// TIA Portal V17 export
// export: Created 2023-02-13T11:16:18.7085922Z, ExportSetting WithDefaults, DisplayName Totally Integrated Automation Portal, DisplayVersion V17, DisplayName TIA Portal Openness, DisplayVersion V17, DisplayName TIA Portal Teamcenter Gateway, DisplayVersion V17, DisplayName TIA Portal Version Control Interface, DisplayVersion V17, DisplayName SINAMICS Startdrive Advanced, DisplayVersion V17, DisplayName SINAMICS Startdrive G130, G150, S120, S150, SINAMICS MV, S210, DisplayVersion V17, DisplayName SINAMICS Startdrive G110M, G120, G120C, G120D, G120P, G115D, DisplayVersion V17, DisplayName STEP 7 Professional, DisplayVersion V17, DisplayName STEP 7 Safety, DisplayVersion V17, DisplayName WinCC Professional, DisplayVersion V17
FUNCTION_BLOCK "IO_Valve_Blend30"   // FB26, LAD
{ S7_Optimized_Access := 'FALSE' }
VERSION : 0.1
// stored: AutoNumber true, IsIECCheckEnabled false, SetENOAutomatically false, UDAEnableTagReadback false
   VAR_INPUT
      "lock 1" : Bool;
      "lock 2" : Bool;
      "lock 3" : Bool;
      "lock 4" : Bool;
      init : Bool;
      reset : Bool;
      testing : Bool;
   END_VAR
   VAR
      "AV-30.01" : "Valve";
      "AV-30.02" : "Valve";
      "AV-30.03" : "Valve";
      "AV-30.04" : "Valve";
      "AV-30.05" : "Valve";
      "AV-30.06" : "Valve";
      "AV-30.07" : "Valve";
      "AV-30.08" : "Valve";
      "AV-30.09" : "Valve";
      "AV-30.10" : "Valve";
      "AV-30.11" : "Valve";
      "AV-30.12" : "Valve";
      "AV-30.13" : "Valve";
      "AV-30.14" : "Valve";
      "AV-30.15" : "Valve";
      "AV-30.16" : "Valve";
      "AV-30.17" : "Valve";
      "AV-30.18" : "Valve";
      "AV-30.19" : "Valve";
      "AV-30.20" : "Valve";
      "AV-30.21" : "Valve";
      "AV-30.22" : "Valve";
      "AV-30.23" : "Valve";
      "AV-30.24" : "Valve";
      "AV-30.25" : "Valve";
      "AV-30.26" : "Valve";
      "AV-30.27" : "Valve";
      "AV-30.28" : "Valve";
      "AV-30.29" : "Valve";
      "AV-30.30" : "Valve";
      "AV-30.31" : "Valve";
      "AV-30.32" : "Valve";
      "AV-30.33" : "Valve";
      "AV-30.34" : "Valve";
      "AV-30.35" : "Valve";
      "AV-30.36" : "Valve";
      "AV-30.41" : "Valve";
      "AV-30.42" : "Valve";
   END_VAR
BEGIN

REGION Network 2 (SCL): FB OPEN AND CLOSE VALVE T-30
   IF #testing THEN
       // Statement section IF
       #"AV-30.01".FB_OPEN := #"AV-30.01".QCMD_OP;
       #"AV-30.01".FB_CLOSE := NOT #"AV-30.01".QCMD_OP;
       #"AV-30.02".FB_OPEN := #"AV-30.02".QCMD_OP;
       #"AV-30.02".FB_CLOSE := NOT #"AV-30.02".QCMD_OP;
       #"AV-30.03".FB_OPEN := #"AV-30.03".QCMD_OP;
       #"AV-30.03".FB_CLOSE := NOT #"AV-30.03".QCMD_OP;
       #"AV-30.04".FB_OPEN := #"AV-30.04".QCMD_OP;
       #"AV-30.04".FB_CLOSE := NOT #"AV-30.04".QCMD_OP;
       #"AV-30.05".FB_OPEN := #"AV-30.05".QCMD_OP;
       #"AV-30.05".FB_CLOSE := NOT #"AV-30.05".QCMD_OP;
       #"AV-30.06".FB_OPEN := #"AV-30.06".QCMD_OP;
       #"AV-30.06".FB_CLOSE := NOT #"AV-30.06".QCMD_OP;
       #"AV-30.07".FB_OPEN := #"AV-30.07".QCMD_OP;
       #"AV-30.07".FB_CLOSE := NOT #"AV-30.07".QCMD_OP;
       #"AV-30.08".FB_OPEN := #"AV-30.08".QCMD_OP;
       #"AV-30.08".FB_CLOSE := NOT #"AV-30.08".QCMD_OP;
       #"AV-30.09".FB_OPEN := #"AV-30.09".QCMD_OP;
       #"AV-30.09".FB_CLOSE := NOT #"AV-30.09".QCMD_OP;
       #"AV-30.10".FB_OPEN := #"AV-30.10".QCMD_OP;
       #"AV-30.10".FB_CLOSE := NOT #"AV-30.10".QCMD_OP;
       #"AV-30.11".FB_OPEN := #"AV-30.11".QCMD_OP;
       #"AV-30.11".FB_CLOSE := NOT #"AV-30.11".QCMD_OP;
       #"AV-30.12".FB_OPEN := #"AV-30.12".QCMD_OP;
       #"AV-30.12".FB_CLOSE := NOT #"AV-30.12".QCMD_OP;
       #"AV-30.13".FB_OPEN := #"AV-30.13".QCMD_OP;
       #"AV-30.13".FB_CLOSE := NOT #"AV-30.13".QCMD_OP;
       #"AV-30.14".FB_OPEN := #"AV-30.14".QCMD_OP;
       #"AV-30.14".FB_CLOSE := NOT #"AV-30.14".QCMD_OP;
       #"AV-30.15".FB_OPEN := #"AV-30.15".QCMD_OP;
       #"AV-30.15".FB_CLOSE := NOT #"AV-30.15".QCMD_OP;
       #"AV-30.16".FB_OPEN := #"AV-30.16".QCMD_OP;
       #"AV-30.16".FB_CLOSE := NOT #"AV-30.16".QCMD_OP;
       #"AV-30.17".FB_OPEN := #"AV-30.17".QCMD_OP;
       #"AV-30.17".FB_CLOSE := NOT #"AV-30.17".QCMD_OP;
       #"AV-30.18".FB_OPEN := #"AV-30.18".QCMD_OP;
       #"AV-30.18".FB_CLOSE := NOT #"AV-30.18".QCMD_OP;
       #"AV-30.19".FB_OPEN := #"AV-30.19".QCMD_OP;
       #"AV-30.19".FB_CLOSE := NOT #"AV-30.19".QCMD_OP;
       #"AV-30.20".FB_OPEN := #"AV-30.20".QCMD_OP;
       #"AV-30.20".FB_CLOSE := NOT #"AV-30.20".QCMD_OP;
       #"AV-30.21".FB_OPEN := #"AV-30.21".QCMD_OP;
       #"AV-30.21".FB_CLOSE := NOT #"AV-30.21".QCMD_OP;
       #"AV-30.22".FB_OPEN := #"AV-30.22".QCMD_OP;
       #"AV-30.22".FB_CLOSE := NOT #"AV-30.22".QCMD_OP;
       #"AV-30.23".FB_OPEN := #"AV-30.23".QCMD_OP;
       #"AV-30.23".FB_CLOSE := NOT #"AV-30.23".QCMD_OP;
       #"AV-30.24".FB_OPEN := #"AV-30.24".QCMD_OP;
       #"AV-30.24".FB_CLOSE := NOT #"AV-30.24".QCMD_OP;
       #"AV-30.25".FB_OPEN := #"AV-30.25".QCMD_OP;
       #"AV-30.25".FB_CLOSE := NOT #"AV-30.25".QCMD_OP;
       #"AV-30.26".FB_OPEN := #"AV-30.26".QCMD_OP;
       #"AV-30.26".FB_CLOSE := NOT #"AV-30.26".QCMD_OP;
       #"AV-30.27".FB_OPEN := #"AV-30.27".QCMD_OP;
       #"AV-30.27".FB_CLOSE := NOT #"AV-30.27".QCMD_OP;
       #"AV-30.28".FB_OPEN := #"AV-30.28".QCMD_OP;
       #"AV-30.28".FB_CLOSE := NOT #"AV-30.28".QCMD_OP;
       #"AV-30.29".FB_OPEN := #"AV-30.29".QCMD_OP;
       #"AV-30.29".FB_CLOSE := NOT #"AV-30.29".QCMD_OP;
       #"AV-30.30".FB_OPEN := #"AV-30.30".QCMD_OP;
       #"AV-30.30".FB_CLOSE := NOT #"AV-30.30".QCMD_OP;
       #"AV-30.31".FB_OPEN := #"AV-30.31".QCMD_OP;
       #"AV-30.31".FB_CLOSE := NOT #"AV-30.31".QCMD_OP;
       #"AV-30.32".FB_OPEN := #"AV-30.32".QCMD_OP;
       #"AV-30.32".FB_CLOSE := NOT #"AV-30.32".QCMD_OP;
       #"AV-30.33".FB_OPEN := #"AV-30.33".QCMD_OP;
       #"AV-30.33".FB_CLOSE := NOT #"AV-30.33".QCMD_OP;
       #"AV-30.34".FB_OPEN := #"AV-30.34".QCMD_OP;
       #"AV-30.34".FB_CLOSE := NOT #"AV-30.34".QCMD_OP;
       #"AV-30.35".FB_OPEN := #"AV-30.35".QCMD_OP;
       #"AV-30.35".FB_CLOSE := NOT #"AV-30.35".QCMD_OP;
       #"AV-30.36".FB_OPEN := #"AV-30.36".QCMD_OP;
       #"AV-30.36".FB_CLOSE := NOT #"AV-30.36".QCMD_OP;
       #"AV-30.41".FB_OPEN := #"AV-30.41".QCMD_OP;
       #"AV-30.41".FB_CLOSE := NOT #"AV-30.41".QCMD_OP;
       #"AV-30.42".FB_OPEN := #"AV-30.42".QCMD_OP;
       #"AV-30.42".FB_CLOSE := NOT #"AV-30.42".QCMD_OP;
   ELSE
       // Statement section ELSE
       #"AV-30.01".FB_OPEN := #"AV-30.01".QCMD_OP;
       #"AV-30.01".FB_CLOSE := NOT #"AV-30.01".QCMD_OP;
       #"AV-30.02".FB_OPEN := NOT "ZSC-30.02";
       #"AV-30.02".FB_CLOSE := "ZSC-30.02";
       #"AV-30.03".FB_OPEN := NOT "ZSC-30.03";
       #"AV-30.03".FB_CLOSE := "ZSC-30.03";
       #"AV-30.04".FB_OPEN := #"AV-30.04".QCMD_OP;
       #"AV-30.04".FB_CLOSE := NOT #"AV-30.04".QCMD_OP;
       #"AV-30.05".FB_OPEN := NOT "ZSC-30.05";
       #"AV-30.05".FB_CLOSE := "ZSC-30.05";
       #"AV-30.06".FB_OPEN := NOT "ZSC-30.06";
       #"AV-30.06".FB_CLOSE := "ZSC-30.06";
       #"AV-30.07".FB_OPEN := #"AV-30.07".QCMD_OP;
       #"AV-30.07".FB_CLOSE := NOT #"AV-30.07".QCMD_OP;
       #"AV-30.08".FB_OPEN := NOT "ZSC-30.08";
       #"AV-30.08".FB_CLOSE := "ZSC-30.08";
       #"AV-30.09".FB_OPEN := NOT "ZSC-30.09";
       #"AV-30.09".FB_CLOSE := "ZSC-30.09";
       #"AV-30.10".FB_OPEN := #"AV-30.10".QCMD_OP;
       #"AV-30.10".FB_CLOSE := NOT #"AV-30.10".QCMD_OP;
       #"AV-30.11".FB_OPEN := NOT "ZSC-30.11";
       #"AV-30.11".FB_CLOSE := "ZSC-30.11";
       #"AV-30.12".FB_OPEN := #"AV-30.12".QCMD_OP;
       #"AV-30.12".FB_CLOSE := NOT #"AV-30.12".QCMD_OP;
       #"AV-30.13".FB_OPEN := #"AV-30.13".QCMD_OP;
       #"AV-30.13".FB_CLOSE := NOT #"AV-30.13".QCMD_OP;
       #"AV-30.14".FB_OPEN := NOT "ZSC-30.14";
       #"AV-30.14".FB_CLOSE := "ZSC-30.14";
       #"AV-30.15".FB_OPEN := #"AV-30.15".QCMD_OP;
       #"AV-30.15".FB_CLOSE := NOT #"AV-30.15".QCMD_OP;
       #"AV-30.16".FB_OPEN := #"AV-30.16".QCMD_OP;
       #"AV-30.16".FB_CLOSE := NOT #"AV-30.16".QCMD_OP;
       #"AV-30.17".FB_OPEN := NOT "ZSC-30.17";
       #"AV-30.17".FB_CLOSE := "ZSC-30.17";
       #"AV-30.18".FB_OPEN := #"AV-30.18".QCMD_OP;
       #"AV-30.18".FB_CLOSE := NOT #"AV-30.18".QCMD_OP;
       #"AV-30.19".FB_OPEN := #"AV-30.19".QCMD_OP;
       #"AV-30.19".FB_CLOSE := NOT #"AV-30.19".QCMD_OP;
       #"AV-30.20".FB_OPEN := NOT "ZSC-30.20";
       #"AV-30.20".FB_CLOSE := "ZSC-30.20";
       #"AV-30.21".FB_OPEN := NOT "ZSC-30.21";
       #"AV-30.21".FB_CLOSE := "ZSC-30.21";
       #"AV-30.22".FB_OPEN := #"AV-30.22".QCMD_OP;
       #"AV-30.22".FB_CLOSE := NOT #"AV-30.22".QCMD_OP;
       #"AV-30.23".FB_OPEN := NOT "ZSC-30.23";
       #"AV-30.23".FB_CLOSE := "ZSC-30.23";
       #"AV-30.24".FB_OPEN := NOT "ZSC-30.24";
       #"AV-30.24".FB_CLOSE := "ZSC-30.24";
       #"AV-30.25".FB_OPEN := NOT "ZSC-30.25";
       #"AV-30.25".FB_CLOSE := "ZSC-30.25";
       #"AV-30.26".FB_OPEN := #"AV-30.26".QCMD_OP;
       #"AV-30.26".FB_CLOSE := NOT #"AV-30.26".QCMD_OP;
       #"AV-30.27".FB_OPEN := NOT "ZSC-30.27";
       #"AV-30.27".FB_CLOSE := "ZSC-30.27";
       #"AV-30.28".FB_OPEN := NOT "ZSC-30.28";
       #"AV-30.28".FB_CLOSE := "ZSC-30.28";
       #"AV-30.29".FB_OPEN := #"AV-30.29".QCMD_OP;
       #"AV-30.29".FB_CLOSE := NOT #"AV-30.29".QCMD_OP;
       #"AV-30.30".FB_OPEN := #"AV-30.30".QCMD_OP;
       #"AV-30.30".FB_CLOSE := NOT #"AV-30.30".QCMD_OP;
       #"AV-30.31".FB_OPEN := NOT "ZSC-30.31";
       #"AV-30.31".FB_CLOSE := "ZSC-30.31";
       #"AV-30.32".FB_OPEN := NOT "ZSC-30.32";
       #"AV-30.32".FB_CLOSE := "ZSC-30.32";
       #"AV-30.33".FB_OPEN := NOT "ZSC-30.33";
       #"AV-30.33".FB_CLOSE := "ZSC-30.33";
       #"AV-30.34".FB_OPEN := NOT "ZSC-30.34";
       #"AV-30.34".FB_CLOSE := "ZSC-30.34";
       #"AV-30.35".FB_OPEN := NOT "ZSC-30.35";
       #"AV-30.35".FB_CLOSE := "ZSC-30.35";
       #"AV-30.36".FB_OPEN := NOT "ZSC-30.36";
       #"AV-30.36".FB_CLOSE := "ZSC-30.36";
       #"AV-30.41".FB_OPEN := #"AV-30.41".QCMD_OP;
       #"AV-30.41".FB_CLOSE := NOT #"AV-30.41".QCMD_OP;
       #"AV-30.42".FB_OPEN := #"AV-30.42".QCMD_OP;
       #"AV-30.42".FB_CLOSE := NOT #"AV-30.42".QCMD_OP;
   END_IF;
END_REGION

NETWORK
TITLE = FB MONITORING TIME VALVE T-30
// FB OPEN TIME
      L     T#20s;
      T     #"AV-30.01".MON_T;
      T     #"AV-30.02".MON_T;
      T     #"AV-30.03".MON_T;
      T     #"AV-30.04".MON_T;
      T     #"AV-30.05".MON_T;
      T     #"AV-30.06".MON_T;
      T     #"AV-30.07".MON_T;
      T     #"AV-30.08".MON_T;
      T     #"AV-30.09".MON_T;
      T     #"AV-30.10".MON_T;
      T     #"AV-30.11".MON_T;
      T     #"AV-30.12".MON_T;
      T     #"AV-30.13".MON_T;
      T     #"AV-30.14".MON_T;
      T     #"AV-30.15".MON_T;
      T     #"AV-30.16".MON_T;
      T     #"AV-30.17".MON_T;
      T     #"AV-30.18".MON_T;
      T     #"AV-30.19".MON_T;
      T     #"AV-30.20".MON_T;
      T     #"AV-30.21".MON_T;
      T     #"AV-30.22".MON_T;
      T     #"AV-30.23".MON_T;
      T     #"AV-30.24".MON_T;
      T     #"AV-30.25".MON_T;
      T     #"AV-30.26".MON_T;
      T     #"AV-30.27".MON_T;
      T     #"AV-30.28".MON_T;
      T     #"AV-30.29".MON_T;
      T     #"AV-30.30".MON_T;
      T     #"AV-30.31".MON_T;
      T     #"AV-30.32".MON_T;
      T     #"AV-30.33".MON_T;
      T     #"AV-30.34".MON_T;
      T     #"AV-30.35".MON_T;
      T     #"AV-30.36".MON_T;
      T     #"AV-30.41".MON_T;
      T     #"AV-30.42".MON_T;
// FB CLOSE TIME
      L     T#20s;
      T     #"AV-30.01".MON_T_CLOSE;
      T     #"AV-30.02".MON_T_CLOSE;
      T     #"AV-30.03".MON_T_CLOSE;
      T     #"AV-30.04".MON_T_CLOSE;
      T     #"AV-30.05".MON_T_CLOSE;
      T     #"AV-30.06".MON_T_CLOSE;
      T     #"AV-30.07".MON_T_CLOSE;
      T     #"AV-30.08".MON_T_CLOSE;
      T     #"AV-30.09".MON_T_CLOSE;
      T     #"AV-30.10".MON_T_CLOSE;
      T     #"AV-30.11".MON_T_CLOSE;
      T     #"AV-30.12".MON_T_CLOSE;
      T     #"AV-30.13".MON_T_CLOSE;
      T     #"AV-30.14".MON_T_CLOSE;
      T     #"AV-30.15".MON_T_CLOSE;
      T     #"AV-30.16".MON_T_CLOSE;
      T     #"AV-30.17".MON_T_CLOSE;
      T     #"AV-30.18".MON_T_CLOSE;
      T     #"AV-30.19".MON_T_CLOSE;
      T     #"AV-30.20".MON_T_CLOSE;
      T     #"AV-30.21".MON_T_CLOSE;
      T     #"AV-30.22".MON_T_CLOSE;
      T     #"AV-30.23".MON_T_CLOSE;
      T     #"AV-30.24".MON_T_CLOSE;
      T     #"AV-30.25".MON_T_CLOSE;
      T     #"AV-30.26".MON_T_CLOSE;
      T     #"AV-30.27".MON_T_CLOSE;
      T     #"AV-30.28".MON_T_CLOSE;
      T     #"AV-30.29".MON_T_CLOSE;
      T     #"AV-30.30".MON_T_CLOSE;
      T     #"AV-30.31".MON_T_CLOSE;
      T     #"AV-30.32".MON_T_CLOSE;
      T     #"AV-30.33".MON_T_CLOSE;
      T     #"AV-30.34".MON_T_CLOSE;
      T     #"AV-30.35".MON_T_CLOSE;
      T     #"AV-30.36".MON_T_CLOSE;
      T     #"AV-30.41".MON_T_CLOSE;
      T     #"AV-30.42".MON_T_CLOSE;

REGION Network 4: AV-30.01
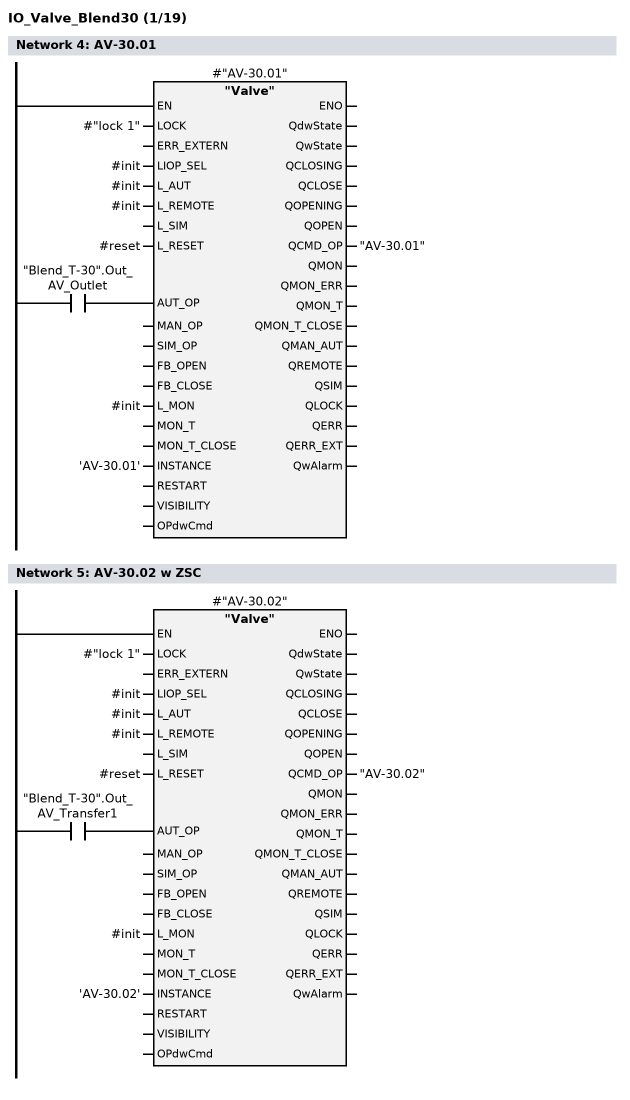
   RUNG wire#powerrail
      #"AV-30.01"(AUT_OP := wire#w1, LOCK := #"lock 1", ERR_EXTERN :=, LIOP_SEL := #init, L_AUT := #init, L_REMOTE := #init, L_SIM :=, L_RESET := #reset, MAN_OP :=, SIM_OP :=, FB_OPEN :=, FB_CLOSE :=, L_MON := #init, MON_T :=, MON_T_CLOSE :=, INSTANCE := 'AV-30.01', RESTART :=, VISIBILITY :=, OPdwCmd :=, QdwState =>, QwState =>, QCLOSING =>, QCLOSE =>, QOPENING =>, QOPEN =>, QCMD_OP => "AV-30.01", QMON =>, QMON_ERR =>, QMON_T =>, QMON_T_CLOSE =>, QMAN_AUT =>, QREMOTE =>, QSIM =>, QLOCK =>, QERR =>, QERR_EXT =>, QwAlarm =>)
   END_RUNG
   RUNG wire#powerrail
      Contact( "Blend_T-30".Out_AV_Outlet )
   END_RUNG wire#w1
   // the same network as SCL:
   #"AV-30.01"(LOCK := #"lock 1",   // "Valve"
               LIOP_SEL := #init,
               L_AUT := #init,
               L_REMOTE := #init,
               L_RESET := #reset,
               AUT_OP := "Blend_T-30".Out_AV_Outlet,
               L_MON := #init,
               INSTANCE := 'AV-30.01',
               QCMD_OP => "AV-30.01");
END_REGION

REGION Network 5: AV-30.02 w ZSC
   RUNG wire#powerrail
      #"AV-30.02"(AUT_OP := wire#w1, LOCK := #"lock 1", ERR_EXTERN :=, LIOP_SEL := #init, L_AUT := #init, L_REMOTE := #init, L_SIM :=, L_RESET := #reset, MAN_OP :=, SIM_OP :=, FB_OPEN :=, FB_CLOSE :=, L_MON := #init, MON_T :=, MON_T_CLOSE :=, INSTANCE := 'AV-30.02', RESTART :=, VISIBILITY :=, OPdwCmd :=, QdwState =>, QwState =>, QCLOSING =>, QCLOSE =>, QOPENING =>, QOPEN =>, QCMD_OP => "AV-30.02", QMON =>, QMON_ERR =>, QMON_T =>, QMON_T_CLOSE =>, QMAN_AUT =>, QREMOTE =>, QSIM =>, QLOCK =>, QERR =>, QERR_EXT =>, QwAlarm =>)
   END_RUNG
   RUNG wire#powerrail
      Contact( "Blend_T-30".Out_AV_Transfer1 )
   END_RUNG wire#w1
   // the same network as SCL:
   #"AV-30.02"(LOCK := #"lock 1",   // "Valve"
               LIOP_SEL := #init,
               L_AUT := #init,
               L_REMOTE := #init,
               L_RESET := #reset,
               AUT_OP := "Blend_T-30".Out_AV_Transfer1,
               L_MON := #init,
               INSTANCE := 'AV-30.02',
               QCMD_OP => "AV-30.02");
END_REGION

REGION Network 6: AV-30.03 w ZSC
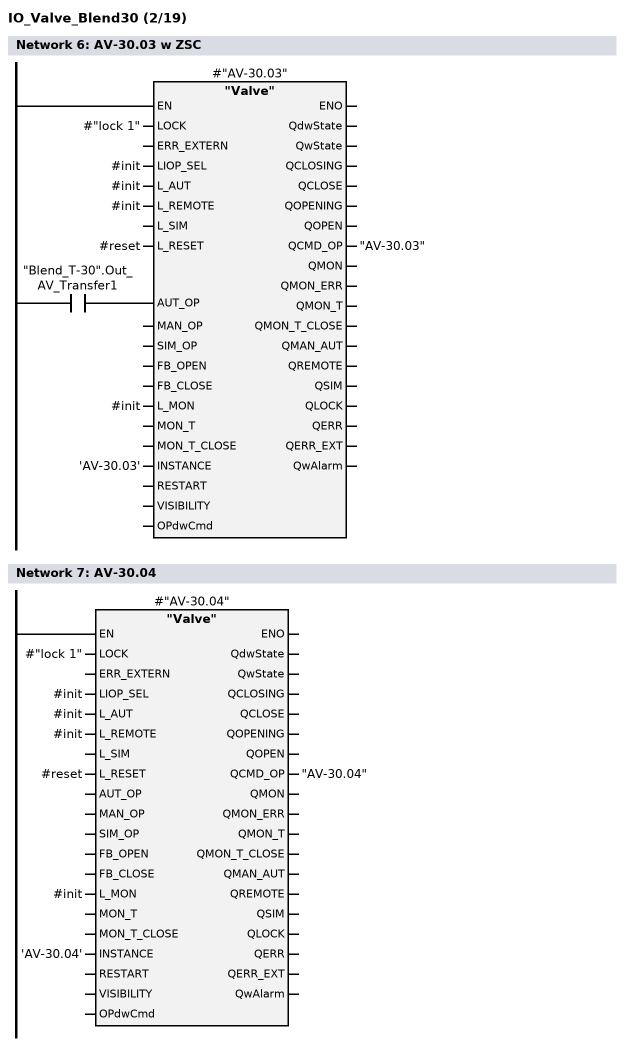
   RUNG wire#powerrail
      #"AV-30.03"(AUT_OP := wire#w1, LOCK := #"lock 1", ERR_EXTERN :=, LIOP_SEL := #init, L_AUT := #init, L_REMOTE := #init, L_SIM :=, L_RESET := #reset, MAN_OP :=, SIM_OP :=, FB_OPEN :=, FB_CLOSE :=, L_MON := #init, MON_T :=, MON_T_CLOSE :=, INSTANCE := 'AV-30.03', RESTART :=, VISIBILITY :=, OPdwCmd :=, QdwState =>, QwState =>, QCLOSING =>, QCLOSE =>, QOPENING =>, QOPEN =>, QCMD_OP => "AV-30.03", QMON =>, QMON_ERR =>, QMON_T =>, QMON_T_CLOSE =>, QMAN_AUT =>, QREMOTE =>, QSIM =>, QLOCK =>, QERR =>, QERR_EXT =>, QwAlarm =>)
   END_RUNG
   RUNG wire#powerrail
      Contact( "Blend_T-30".Out_AV_Transfer1 )
   END_RUNG wire#w1
   // the same network as SCL:
   #"AV-30.03"(LOCK := #"lock 1",   // "Valve"
               LIOP_SEL := #init,
               L_AUT := #init,
               L_REMOTE := #init,
               L_RESET := #reset,
               AUT_OP := "Blend_T-30".Out_AV_Transfer1,
               L_MON := #init,
               INSTANCE := 'AV-30.03',
               QCMD_OP => "AV-30.03");
END_REGION

REGION Network 7: AV-30.04
   RUNG wire#powerrail
      #"AV-30.04"(LOCK := #"lock 1", ERR_EXTERN :=, LIOP_SEL := #init, L_AUT := #init, L_REMOTE := #init, L_SIM :=, L_RESET := #reset, AUT_OP :=, MAN_OP :=, SIM_OP :=, FB_OPEN :=, FB_CLOSE :=, L_MON := #init, MON_T :=, MON_T_CLOSE :=, INSTANCE := 'AV-30.04', RESTART :=, VISIBILITY :=, OPdwCmd :=, QdwState =>, QwState =>, QCLOSING =>, QCLOSE =>, QOPENING =>, QOPEN =>, QCMD_OP => "AV-30.04", QMON =>, QMON_ERR =>, QMON_T =>, QMON_T_CLOSE =>, QMAN_AUT =>, QREMOTE =>, QSIM =>, QLOCK =>, QERR =>, QERR_EXT =>, QwAlarm =>)
   END_RUNG
   // the same network as SCL:
   #"AV-30.04"(LOCK := #"lock 1",   // "Valve"
               LIOP_SEL := #init,
               L_AUT := #init,
               L_REMOTE := #init,
               L_RESET := #reset,
               L_MON := #init,
               INSTANCE := 'AV-30.04',
               QCMD_OP => "AV-30.04");
END_REGION

REGION Network 8: AV-30.05 w ZSC
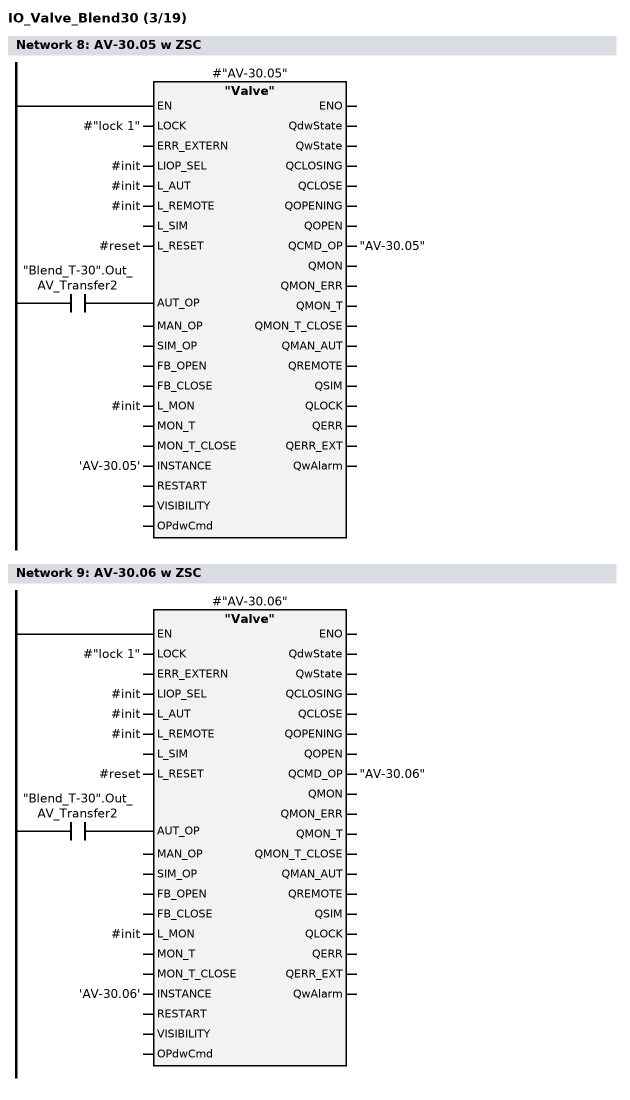
   RUNG wire#powerrail
      #"AV-30.05"(AUT_OP := wire#w1, LOCK := #"lock 1", ERR_EXTERN :=, LIOP_SEL := #init, L_AUT := #init, L_REMOTE := #init, L_SIM :=, L_RESET := #reset, MAN_OP :=, SIM_OP :=, FB_OPEN :=, FB_CLOSE :=, L_MON := #init, MON_T :=, MON_T_CLOSE :=, INSTANCE := 'AV-30.05', RESTART :=, VISIBILITY :=, OPdwCmd :=, QdwState =>, QwState =>, QCLOSING =>, QCLOSE =>, QOPENING =>, QOPEN =>, QCMD_OP => "AV-30.05", QMON =>, QMON_ERR =>, QMON_T =>, QMON_T_CLOSE =>, QMAN_AUT =>, QREMOTE =>, QSIM =>, QLOCK =>, QERR =>, QERR_EXT =>, QwAlarm =>)
   END_RUNG
   RUNG wire#powerrail
      Contact( "Blend_T-30".Out_AV_Transfer2 )
   END_RUNG wire#w1
   // the same network as SCL:
   #"AV-30.05"(LOCK := #"lock 1",   // "Valve"
               LIOP_SEL := #init,
               L_AUT := #init,
               L_REMOTE := #init,
               L_RESET := #reset,
               AUT_OP := "Blend_T-30".Out_AV_Transfer2,
               L_MON := #init,
               INSTANCE := 'AV-30.05',
               QCMD_OP => "AV-30.05");
END_REGION

REGION Network 9: AV-30.06 w ZSC
   RUNG wire#powerrail
      #"AV-30.06"(AUT_OP := wire#w1, LOCK := #"lock 1", ERR_EXTERN :=, LIOP_SEL := #init, L_AUT := #init, L_REMOTE := #init, L_SIM :=, L_RESET := #reset, MAN_OP :=, SIM_OP :=, FB_OPEN :=, FB_CLOSE :=, L_MON := #init, MON_T :=, MON_T_CLOSE :=, INSTANCE := 'AV-30.06', RESTART :=, VISIBILITY :=, OPdwCmd :=, QdwState =>, QwState =>, QCLOSING =>, QCLOSE =>, QOPENING =>, QOPEN =>, QCMD_OP => "AV-30.06", QMON =>, QMON_ERR =>, QMON_T =>, QMON_T_CLOSE =>, QMAN_AUT =>, QREMOTE =>, QSIM =>, QLOCK =>, QERR =>, QERR_EXT =>, QwAlarm =>)
   END_RUNG
   RUNG wire#powerrail
      Contact( "Blend_T-30".Out_AV_Transfer2 )
   END_RUNG wire#w1
   // the same network as SCL:
   #"AV-30.06"(LOCK := #"lock 1",   // "Valve"
               LIOP_SEL := #init,
               L_AUT := #init,
               L_REMOTE := #init,
               L_RESET := #reset,
               AUT_OP := "Blend_T-30".Out_AV_Transfer2,
               L_MON := #init,
               INSTANCE := 'AV-30.06',
               QCMD_OP => "AV-30.06");
END_REGION

REGION Network 10: AV-30.07
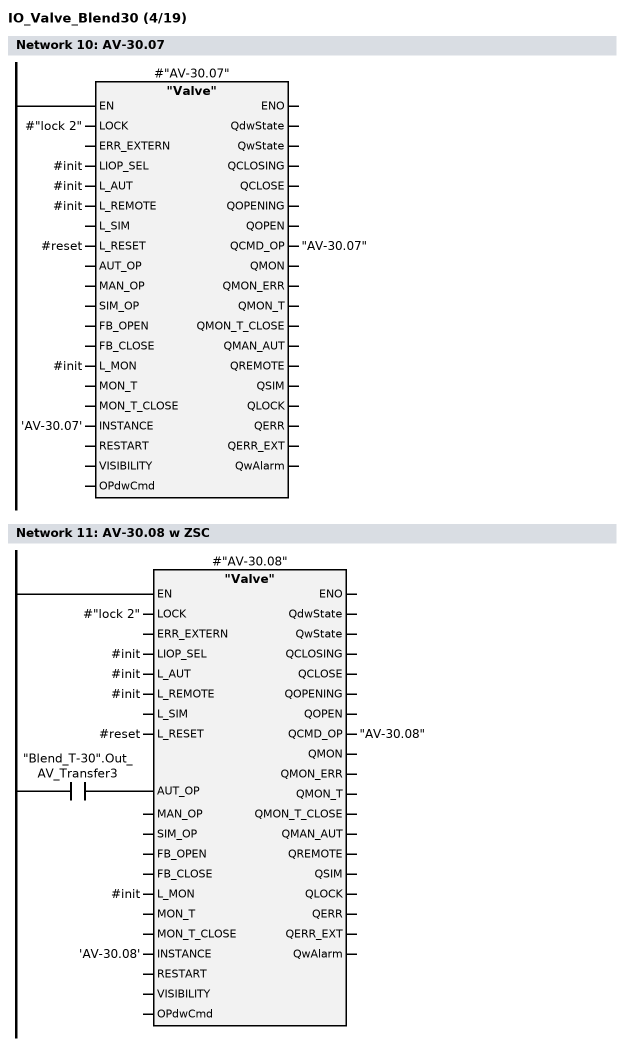
   RUNG wire#powerrail
      #"AV-30.07"(LOCK := #"lock 2", ERR_EXTERN :=, LIOP_SEL := #init, L_AUT := #init, L_REMOTE := #init, L_SIM :=, L_RESET := #reset, AUT_OP :=, MAN_OP :=, SIM_OP :=, FB_OPEN :=, FB_CLOSE :=, L_MON := #init, MON_T :=, MON_T_CLOSE :=, INSTANCE := 'AV-30.07', RESTART :=, VISIBILITY :=, OPdwCmd :=, QdwState =>, QwState =>, QCLOSING =>, QCLOSE =>, QOPENING =>, QOPEN =>, QCMD_OP => "AV-30.07", QMON =>, QMON_ERR =>, QMON_T =>, QMON_T_CLOSE =>, QMAN_AUT =>, QREMOTE =>, QSIM =>, QLOCK =>, QERR =>, QERR_EXT =>, QwAlarm =>)
   END_RUNG
   // the same network as SCL:
   #"AV-30.07"(LOCK := #"lock 2",   // "Valve"
               LIOP_SEL := #init,
               L_AUT := #init,
               L_REMOTE := #init,
               L_RESET := #reset,
               L_MON := #init,
               INSTANCE := 'AV-30.07',
               QCMD_OP => "AV-30.07");
END_REGION

REGION Network 11: AV-30.08 w ZSC
   RUNG wire#powerrail
      #"AV-30.08"(AUT_OP := wire#w1, LOCK := #"lock 2", ERR_EXTERN :=, LIOP_SEL := #init, L_AUT := #init, L_REMOTE := #init, L_SIM :=, L_RESET := #reset, MAN_OP :=, SIM_OP :=, FB_OPEN :=, FB_CLOSE :=, L_MON := #init, MON_T :=, MON_T_CLOSE :=, INSTANCE := 'AV-30.08', RESTART :=, VISIBILITY :=, OPdwCmd :=, QdwState =>, QwState =>, QCLOSING =>, QCLOSE =>, QOPENING =>, QOPEN =>, QCMD_OP => "AV-30.08", QMON =>, QMON_ERR =>, QMON_T =>, QMON_T_CLOSE =>, QMAN_AUT =>, QREMOTE =>, QSIM =>, QLOCK =>, QERR =>, QERR_EXT =>, QwAlarm =>)
   END_RUNG
   RUNG wire#powerrail
      Contact( "Blend_T-30".Out_AV_Transfer3 )
   END_RUNG wire#w1
   // the same network as SCL:
   #"AV-30.08"(LOCK := #"lock 2",   // "Valve"
               LIOP_SEL := #init,
               L_AUT := #init,
               L_REMOTE := #init,
               L_RESET := #reset,
               AUT_OP := "Blend_T-30".Out_AV_Transfer3,
               L_MON := #init,
               INSTANCE := 'AV-30.08',
               QCMD_OP => "AV-30.08");
END_REGION

REGION Network 12: AV-30.09 w ZSC
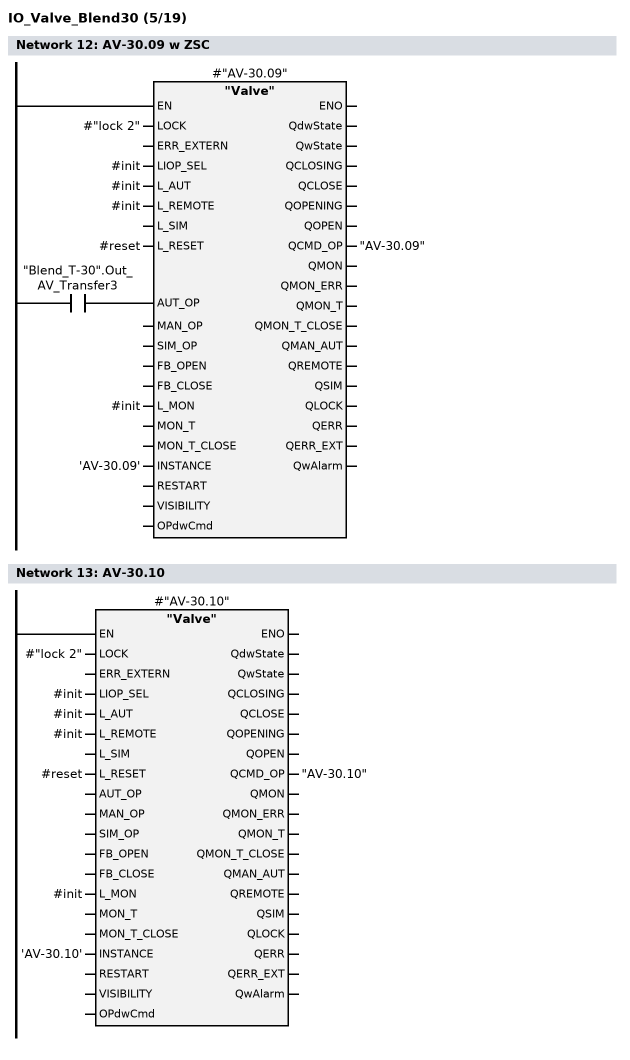
   RUNG wire#powerrail
      #"AV-30.09"(AUT_OP := wire#w1, LOCK := #"lock 2", ERR_EXTERN :=, LIOP_SEL := #init, L_AUT := #init, L_REMOTE := #init, L_SIM :=, L_RESET := #reset, MAN_OP :=, SIM_OP :=, FB_OPEN :=, FB_CLOSE :=, L_MON := #init, MON_T :=, MON_T_CLOSE :=, INSTANCE := 'AV-30.09', RESTART :=, VISIBILITY :=, OPdwCmd :=, QdwState =>, QwState =>, QCLOSING =>, QCLOSE =>, QOPENING =>, QOPEN =>, QCMD_OP => "AV-30.09", QMON =>, QMON_ERR =>, QMON_T =>, QMON_T_CLOSE =>, QMAN_AUT =>, QREMOTE =>, QSIM =>, QLOCK =>, QERR =>, QERR_EXT =>, QwAlarm =>)
   END_RUNG
   RUNG wire#powerrail
      Contact( "Blend_T-30".Out_AV_Transfer3 )
   END_RUNG wire#w1
   // the same network as SCL:
   #"AV-30.09"(LOCK := #"lock 2",   // "Valve"
               LIOP_SEL := #init,
               L_AUT := #init,
               L_REMOTE := #init,
               L_RESET := #reset,
               AUT_OP := "Blend_T-30".Out_AV_Transfer3,
               L_MON := #init,
               INSTANCE := 'AV-30.09',
               QCMD_OP => "AV-30.09");
END_REGION

REGION Network 13: AV-30.10
   RUNG wire#powerrail
      #"AV-30.10"(LOCK := #"lock 2", ERR_EXTERN :=, LIOP_SEL := #init, L_AUT := #init, L_REMOTE := #init, L_SIM :=, L_RESET := #reset, AUT_OP :=, MAN_OP :=, SIM_OP :=, FB_OPEN :=, FB_CLOSE :=, L_MON := #init, MON_T :=, MON_T_CLOSE :=, INSTANCE := 'AV-30.10', RESTART :=, VISIBILITY :=, OPdwCmd :=, QdwState =>, QwState =>, QCLOSING =>, QCLOSE =>, QOPENING =>, QOPEN =>, QCMD_OP => "AV-30.10", QMON =>, QMON_ERR =>, QMON_T =>, QMON_T_CLOSE =>, QMAN_AUT =>, QREMOTE =>, QSIM =>, QLOCK =>, QERR =>, QERR_EXT =>, QwAlarm =>)
   END_RUNG
   // the same network as SCL:
   #"AV-30.10"(LOCK := #"lock 2",   // "Valve"
               LIOP_SEL := #init,
               L_AUT := #init,
               L_REMOTE := #init,
               L_RESET := #reset,
               L_MON := #init,
               INSTANCE := 'AV-30.10',
               QCMD_OP => "AV-30.10");
END_REGION

REGION Network 14: AV-30.11 w ZSC
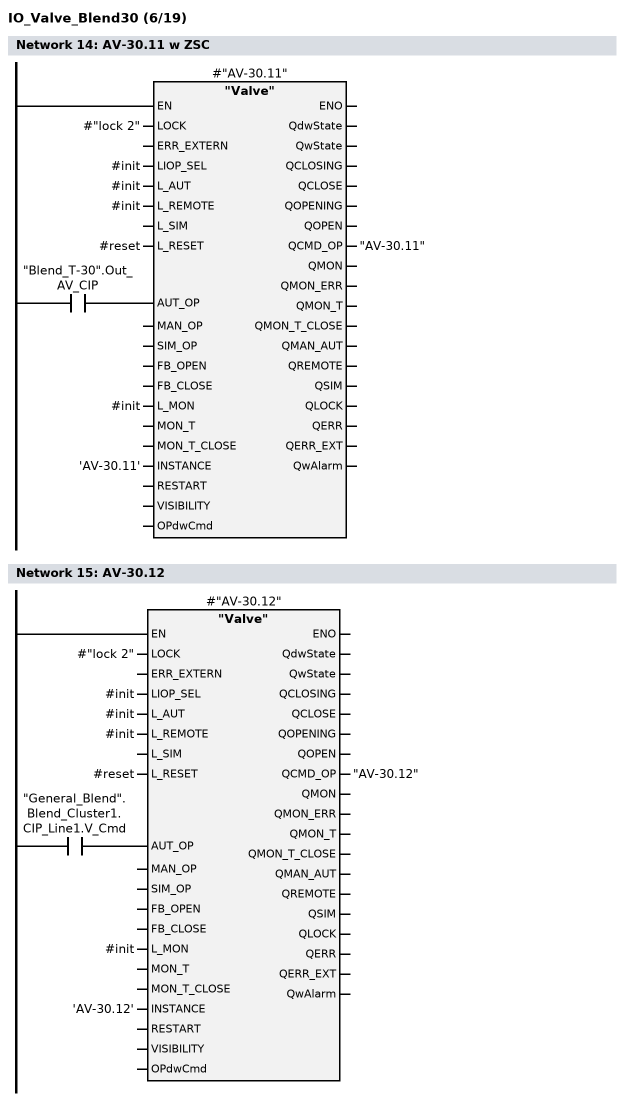
   RUNG wire#powerrail
      #"AV-30.11"(AUT_OP := wire#w1, LOCK := #"lock 2", ERR_EXTERN :=, LIOP_SEL := #init, L_AUT := #init, L_REMOTE := #init, L_SIM :=, L_RESET := #reset, MAN_OP :=, SIM_OP :=, FB_OPEN :=, FB_CLOSE :=, L_MON := #init, MON_T :=, MON_T_CLOSE :=, INSTANCE := 'AV-30.11', RESTART :=, VISIBILITY :=, OPdwCmd :=, QdwState =>, QwState =>, QCLOSING =>, QCLOSE =>, QOPENING =>, QOPEN =>, QCMD_OP => "AV-30.11", QMON =>, QMON_ERR =>, QMON_T =>, QMON_T_CLOSE =>, QMAN_AUT =>, QREMOTE =>, QSIM =>, QLOCK =>, QERR =>, QERR_EXT =>, QwAlarm =>)
   END_RUNG
   RUNG wire#powerrail
      Contact( "Blend_T-30".Out_AV_CIP )
   END_RUNG wire#w1
   // the same network as SCL:
   #"AV-30.11"(LOCK := #"lock 2",   // "Valve"
               LIOP_SEL := #init,
               L_AUT := #init,
               L_REMOTE := #init,
               L_RESET := #reset,
               AUT_OP := "Blend_T-30".Out_AV_CIP,
               L_MON := #init,
               INSTANCE := 'AV-30.11',
               QCMD_OP => "AV-30.11");
END_REGION

REGION Network 15: AV-30.12
   RUNG wire#powerrail
      #"AV-30.12"(AUT_OP := wire#w1, LOCK := #"lock 2", ERR_EXTERN :=, LIOP_SEL := #init, L_AUT := #init, L_REMOTE := #init, L_SIM :=, L_RESET := #reset, MAN_OP :=, SIM_OP :=, FB_OPEN :=, FB_CLOSE :=, L_MON := #init, MON_T :=, MON_T_CLOSE :=, INSTANCE := 'AV-30.12', RESTART :=, VISIBILITY :=, OPdwCmd :=, QdwState =>, QwState =>, QCLOSING =>, QCLOSE =>, QOPENING =>, QOPEN =>, QCMD_OP => "AV-30.12", QMON =>, QMON_ERR =>, QMON_T =>, QMON_T_CLOSE =>, QMAN_AUT =>, QREMOTE =>, QSIM =>, QLOCK =>, QERR =>, QERR_EXT =>, QwAlarm =>)
   END_RUNG
   RUNG wire#powerrail
      Contact( "General_Blend".Blend_Cluster1.CIP_Line1.V_Cmd )
   END_RUNG wire#w1
   // the same network as SCL:
   #"AV-30.12"(LOCK := #"lock 2",   // "Valve"
               LIOP_SEL := #init,
               L_AUT := #init,
               L_REMOTE := #init,
               L_RESET := #reset,
               AUT_OP := "General_Blend".Blend_Cluster1.CIP_Line1.V_Cmd,
               L_MON := #init,
               INSTANCE := 'AV-30.12',
               QCMD_OP => "AV-30.12");
END_REGION

REGION Network 16: AV-30.13
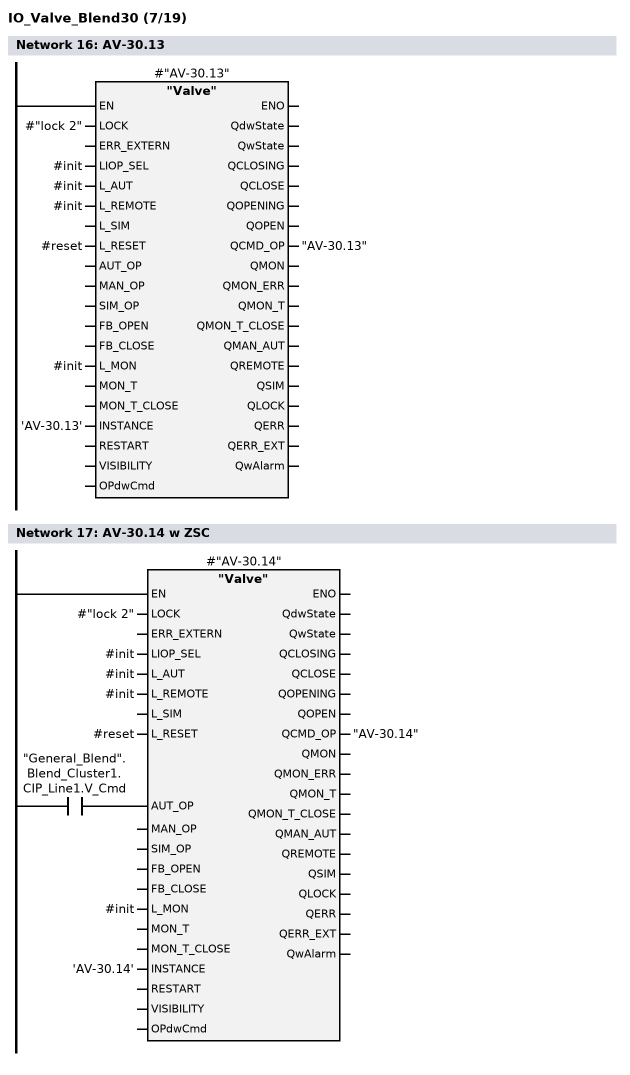
   RUNG wire#powerrail
      #"AV-30.13"(LOCK := #"lock 2", ERR_EXTERN :=, LIOP_SEL := #init, L_AUT := #init, L_REMOTE := #init, L_SIM :=, L_RESET := #reset, AUT_OP :=, MAN_OP :=, SIM_OP :=, FB_OPEN :=, FB_CLOSE :=, L_MON := #init, MON_T :=, MON_T_CLOSE :=, INSTANCE := 'AV-30.13', RESTART :=, VISIBILITY :=, OPdwCmd :=, QdwState =>, QwState =>, QCLOSING =>, QCLOSE =>, QOPENING =>, QOPEN =>, QCMD_OP => "AV-30.13", QMON =>, QMON_ERR =>, QMON_T =>, QMON_T_CLOSE =>, QMAN_AUT =>, QREMOTE =>, QSIM =>, QLOCK =>, QERR =>, QERR_EXT =>, QwAlarm =>)
   END_RUNG
   // the same network as SCL:
   #"AV-30.13"(LOCK := #"lock 2",   // "Valve"
               LIOP_SEL := #init,
               L_AUT := #init,
               L_REMOTE := #init,
               L_RESET := #reset,
               L_MON := #init,
               INSTANCE := 'AV-30.13',
               QCMD_OP => "AV-30.13");
END_REGION

REGION Network 17: AV-30.14 w ZSC
   RUNG wire#powerrail
      #"AV-30.14"(AUT_OP := wire#w1, LOCK := #"lock 2", ERR_EXTERN :=, LIOP_SEL := #init, L_AUT := #init, L_REMOTE := #init, L_SIM :=, L_RESET := #reset, MAN_OP :=, SIM_OP :=, FB_OPEN :=, FB_CLOSE :=, L_MON := #init, MON_T :=, MON_T_CLOSE :=, INSTANCE := 'AV-30.14', RESTART :=, VISIBILITY :=, OPdwCmd :=, QdwState =>, QwState =>, QCLOSING =>, QCLOSE =>, QOPENING =>, QOPEN =>, QCMD_OP => "AV-30.14", QMON =>, QMON_ERR =>, QMON_T =>, QMON_T_CLOSE =>, QMAN_AUT =>, QREMOTE =>, QSIM =>, QLOCK =>, QERR =>, QERR_EXT =>, QwAlarm =>)
   END_RUNG
   RUNG wire#powerrail
      Contact( "General_Blend".Blend_Cluster1.CIP_Line1.V_Cmd )
   END_RUNG wire#w1
   // the same network as SCL:
   #"AV-30.14"(LOCK := #"lock 2",   // "Valve"
               LIOP_SEL := #init,
               L_AUT := #init,
               L_REMOTE := #init,
               L_RESET := #reset,
               AUT_OP := "General_Blend".Blend_Cluster1.CIP_Line1.V_Cmd,
               L_MON := #init,
               INSTANCE := 'AV-30.14',
               QCMD_OP => "AV-30.14");
END_REGION

REGION Network 18: AV-30.15
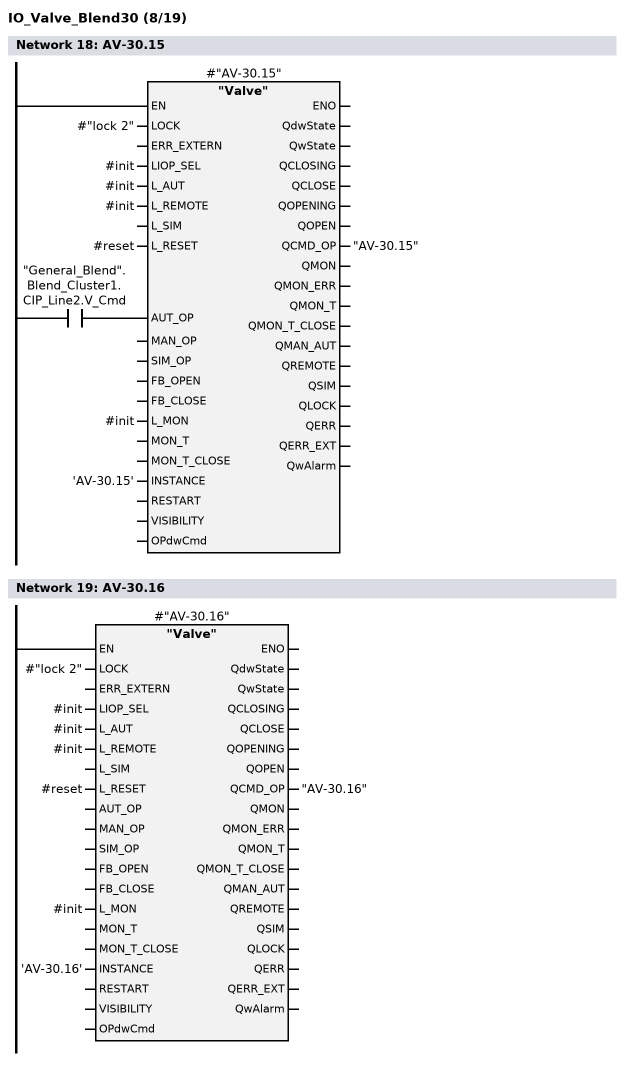
   RUNG wire#powerrail
      #"AV-30.15"(AUT_OP := wire#w1, LOCK := #"lock 2", ERR_EXTERN :=, LIOP_SEL := #init, L_AUT := #init, L_REMOTE := #init, L_SIM :=, L_RESET := #reset, MAN_OP :=, SIM_OP :=, FB_OPEN :=, FB_CLOSE :=, L_MON := #init, MON_T :=, MON_T_CLOSE :=, INSTANCE := 'AV-30.15', RESTART :=, VISIBILITY :=, OPdwCmd :=, QdwState =>, QwState =>, QCLOSING =>, QCLOSE =>, QOPENING =>, QOPEN =>, QCMD_OP => "AV-30.15", QMON =>, QMON_ERR =>, QMON_T =>, QMON_T_CLOSE =>, QMAN_AUT =>, QREMOTE =>, QSIM =>, QLOCK =>, QERR =>, QERR_EXT =>, QwAlarm =>)
   END_RUNG
   RUNG wire#powerrail
      Contact( "General_Blend".Blend_Cluster1.CIP_Line2.V_Cmd )
   END_RUNG wire#w1
   // the same network as SCL:
   #"AV-30.15"(LOCK := #"lock 2",   // "Valve"
               LIOP_SEL := #init,
               L_AUT := #init,
               L_REMOTE := #init,
               L_RESET := #reset,
               AUT_OP := "General_Blend".Blend_Cluster1.CIP_Line2.V_Cmd,
               L_MON := #init,
               INSTANCE := 'AV-30.15',
               QCMD_OP => "AV-30.15");
END_REGION

REGION Network 19: AV-30.16
   RUNG wire#powerrail
      #"AV-30.16"(LOCK := #"lock 2", ERR_EXTERN :=, LIOP_SEL := #init, L_AUT := #init, L_REMOTE := #init, L_SIM :=, L_RESET := #reset, AUT_OP :=, MAN_OP :=, SIM_OP :=, FB_OPEN :=, FB_CLOSE :=, L_MON := #init, MON_T :=, MON_T_CLOSE :=, INSTANCE := 'AV-30.16', RESTART :=, VISIBILITY :=, OPdwCmd :=, QdwState =>, QwState =>, QCLOSING =>, QCLOSE =>, QOPENING =>, QOPEN =>, QCMD_OP => "AV-30.16", QMON =>, QMON_ERR =>, QMON_T =>, QMON_T_CLOSE =>, QMAN_AUT =>, QREMOTE =>, QSIM =>, QLOCK =>, QERR =>, QERR_EXT =>, QwAlarm =>)
   END_RUNG
   // the same network as SCL:
   #"AV-30.16"(LOCK := #"lock 2",   // "Valve"
               LIOP_SEL := #init,
               L_AUT := #init,
               L_REMOTE := #init,
               L_RESET := #reset,
               L_MON := #init,
               INSTANCE := 'AV-30.16',
               QCMD_OP => "AV-30.16");
END_REGION

REGION Network 20: AV-30.17 w ZSC
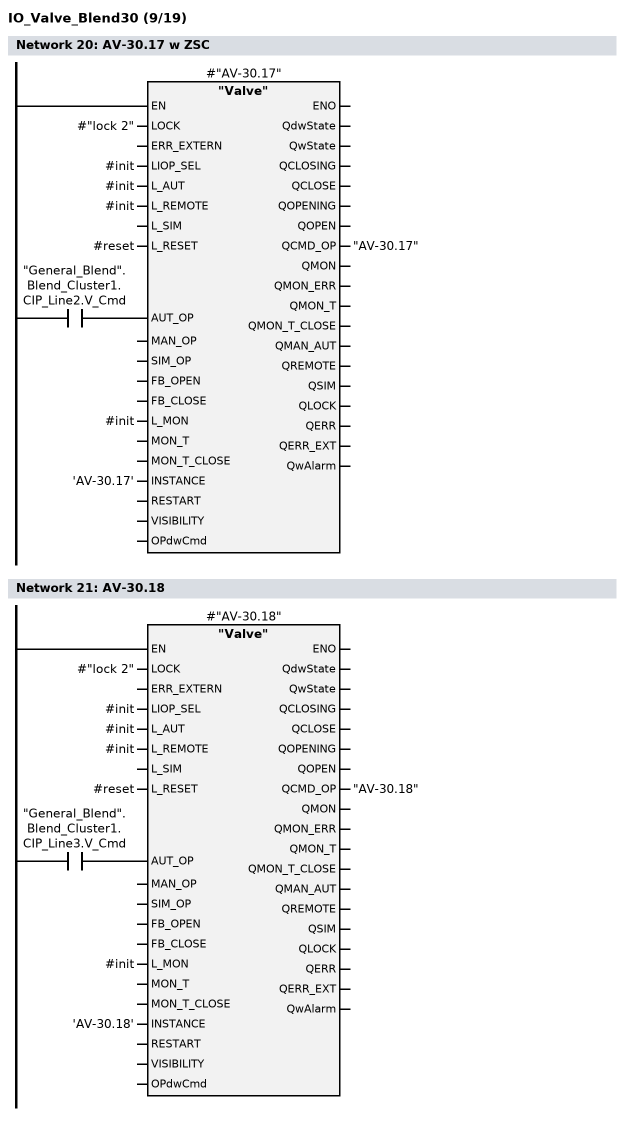
   RUNG wire#powerrail
      #"AV-30.17"(AUT_OP := wire#w1, LOCK := #"lock 2", ERR_EXTERN :=, LIOP_SEL := #init, L_AUT := #init, L_REMOTE := #init, L_SIM :=, L_RESET := #reset, MAN_OP :=, SIM_OP :=, FB_OPEN :=, FB_CLOSE :=, L_MON := #init, MON_T :=, MON_T_CLOSE :=, INSTANCE := 'AV-30.17', RESTART :=, VISIBILITY :=, OPdwCmd :=, QdwState =>, QwState =>, QCLOSING =>, QCLOSE =>, QOPENING =>, QOPEN =>, QCMD_OP => "AV-30.17", QMON =>, QMON_ERR =>, QMON_T =>, QMON_T_CLOSE =>, QMAN_AUT =>, QREMOTE =>, QSIM =>, QLOCK =>, QERR =>, QERR_EXT =>, QwAlarm =>)
   END_RUNG
   RUNG wire#powerrail
      Contact( "General_Blend".Blend_Cluster1.CIP_Line2.V_Cmd )
   END_RUNG wire#w1
   // the same network as SCL:
   #"AV-30.17"(LOCK := #"lock 2",   // "Valve"
               LIOP_SEL := #init,
               L_AUT := #init,
               L_REMOTE := #init,
               L_RESET := #reset,
               AUT_OP := "General_Blend".Blend_Cluster1.CIP_Line2.V_Cmd,
               L_MON := #init,
               INSTANCE := 'AV-30.17',
               QCMD_OP => "AV-30.17");
END_REGION

REGION Network 21: AV-30.18
   RUNG wire#powerrail
      #"AV-30.18"(AUT_OP := wire#w1, LOCK := #"lock 2", ERR_EXTERN :=, LIOP_SEL := #init, L_AUT := #init, L_REMOTE := #init, L_SIM :=, L_RESET := #reset, MAN_OP :=, SIM_OP :=, FB_OPEN :=, FB_CLOSE :=, L_MON := #init, MON_T :=, MON_T_CLOSE :=, INSTANCE := 'AV-30.18', RESTART :=, VISIBILITY :=, OPdwCmd :=, QdwState =>, QwState =>, QCLOSING =>, QCLOSE =>, QOPENING =>, QOPEN =>, QCMD_OP => "AV-30.18", QMON =>, QMON_ERR =>, QMON_T =>, QMON_T_CLOSE =>, QMAN_AUT =>, QREMOTE =>, QSIM =>, QLOCK =>, QERR =>, QERR_EXT =>, QwAlarm =>)
   END_RUNG
   RUNG wire#powerrail
      Contact( "General_Blend".Blend_Cluster1.CIP_Line3.V_Cmd )
   END_RUNG wire#w1
   // the same network as SCL:
   #"AV-30.18"(LOCK := #"lock 2",   // "Valve"
               LIOP_SEL := #init,
               L_AUT := #init,
               L_REMOTE := #init,
               L_RESET := #reset,
               AUT_OP := "General_Blend".Blend_Cluster1.CIP_Line3.V_Cmd,
               L_MON := #init,
               INSTANCE := 'AV-30.18',
               QCMD_OP => "AV-30.18");
END_REGION

REGION Network 22: AV-30.19
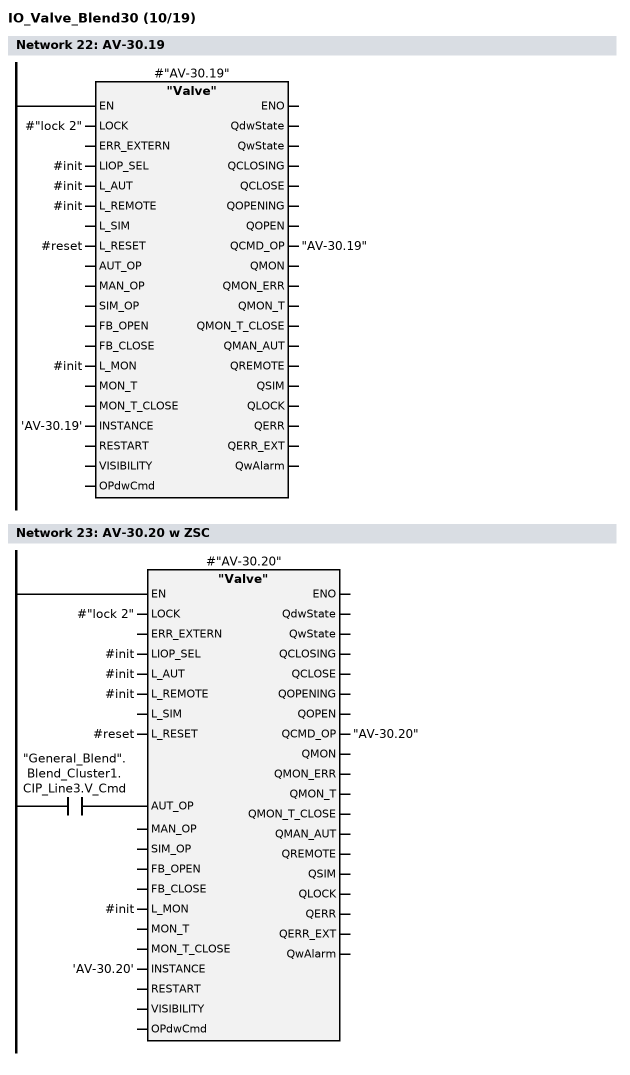
   RUNG wire#powerrail
      #"AV-30.19"(LOCK := #"lock 2", ERR_EXTERN :=, LIOP_SEL := #init, L_AUT := #init, L_REMOTE := #init, L_SIM :=, L_RESET := #reset, AUT_OP :=, MAN_OP :=, SIM_OP :=, FB_OPEN :=, FB_CLOSE :=, L_MON := #init, MON_T :=, MON_T_CLOSE :=, INSTANCE := 'AV-30.19', RESTART :=, VISIBILITY :=, OPdwCmd :=, QdwState =>, QwState =>, QCLOSING =>, QCLOSE =>, QOPENING =>, QOPEN =>, QCMD_OP => "AV-30.19", QMON =>, QMON_ERR =>, QMON_T =>, QMON_T_CLOSE =>, QMAN_AUT =>, QREMOTE =>, QSIM =>, QLOCK =>, QERR =>, QERR_EXT =>, QwAlarm =>)
   END_RUNG
   // the same network as SCL:
   #"AV-30.19"(LOCK := #"lock 2",   // "Valve"
               LIOP_SEL := #init,
               L_AUT := #init,
               L_REMOTE := #init,
               L_RESET := #reset,
               L_MON := #init,
               INSTANCE := 'AV-30.19',
               QCMD_OP => "AV-30.19");
END_REGION

REGION Network 23: AV-30.20 w ZSC
   RUNG wire#powerrail
      #"AV-30.20"(AUT_OP := wire#w1, LOCK := #"lock 2", ERR_EXTERN :=, LIOP_SEL := #init, L_AUT := #init, L_REMOTE := #init, L_SIM :=, L_RESET := #reset, MAN_OP :=, SIM_OP :=, FB_OPEN :=, FB_CLOSE :=, L_MON := #init, MON_T :=, MON_T_CLOSE :=, INSTANCE := 'AV-30.20', RESTART :=, VISIBILITY :=, OPdwCmd :=, QdwState =>, QwState =>, QCLOSING =>, QCLOSE =>, QOPENING =>, QOPEN =>, QCMD_OP => "AV-30.20", QMON =>, QMON_ERR =>, QMON_T =>, QMON_T_CLOSE =>, QMAN_AUT =>, QREMOTE =>, QSIM =>, QLOCK =>, QERR =>, QERR_EXT =>, QwAlarm =>)
   END_RUNG
   RUNG wire#powerrail
      Contact( "General_Blend".Blend_Cluster1.CIP_Line3.V_Cmd )
   END_RUNG wire#w1
   // the same network as SCL:
   #"AV-30.20"(LOCK := #"lock 2",   // "Valve"
               LIOP_SEL := #init,
               L_AUT := #init,
               L_REMOTE := #init,
               L_RESET := #reset,
               AUT_OP := "General_Blend".Blend_Cluster1.CIP_Line3.V_Cmd,
               L_MON := #init,
               INSTANCE := 'AV-30.20',
               QCMD_OP => "AV-30.20");
END_REGION

REGION Network 24: AV-30.21 w ZSC
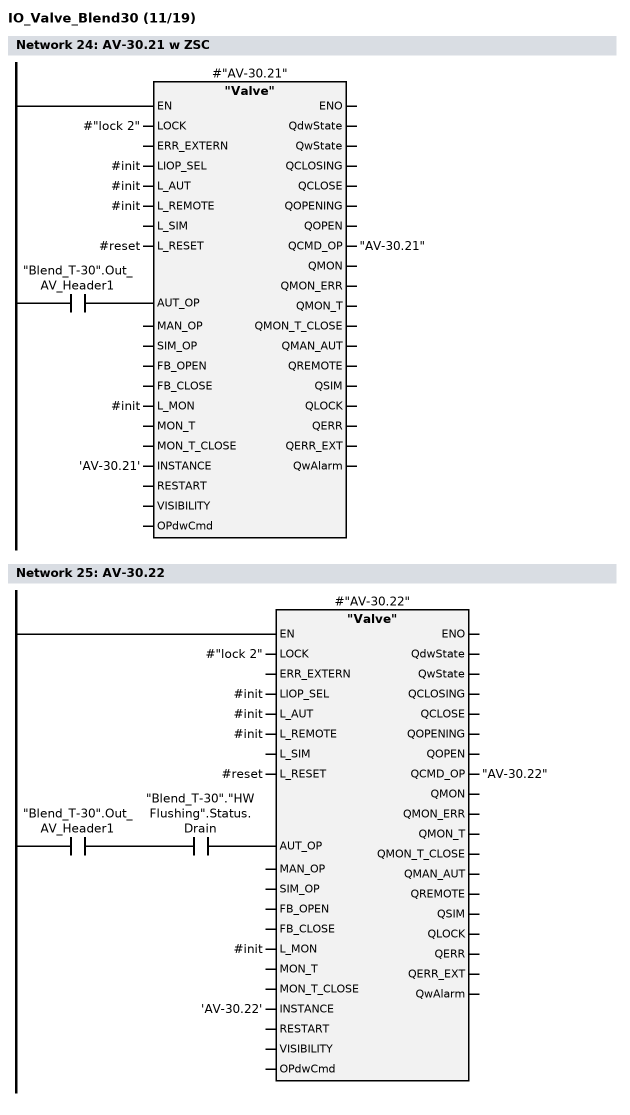
   RUNG wire#powerrail
      #"AV-30.21"(AUT_OP := wire#w1, LOCK := #"lock 2", ERR_EXTERN :=, LIOP_SEL := #init, L_AUT := #init, L_REMOTE := #init, L_SIM :=, L_RESET := #reset, MAN_OP :=, SIM_OP :=, FB_OPEN :=, FB_CLOSE :=, L_MON := #init, MON_T :=, MON_T_CLOSE :=, INSTANCE := 'AV-30.21', RESTART :=, VISIBILITY :=, OPdwCmd :=, QdwState =>, QwState =>, QCLOSING =>, QCLOSE =>, QOPENING =>, QOPEN =>, QCMD_OP => "AV-30.21", QMON =>, QMON_ERR =>, QMON_T =>, QMON_T_CLOSE =>, QMAN_AUT =>, QREMOTE =>, QSIM =>, QLOCK =>, QERR =>, QERR_EXT =>, QwAlarm =>)
   END_RUNG
   RUNG wire#powerrail
      Contact( "Blend_T-30".Out_AV_Header1 )
   END_RUNG wire#w1
   // the same network as SCL:
   #"AV-30.21"(LOCK := #"lock 2",   // "Valve"
               LIOP_SEL := #init,
               L_AUT := #init,
               L_REMOTE := #init,
               L_RESET := #reset,
               AUT_OP := "Blend_T-30".Out_AV_Header1,
               L_MON := #init,
               INSTANCE := 'AV-30.21',
               QCMD_OP => "AV-30.21");
END_REGION

REGION Network 25: AV-30.22
   RUNG wire#powerrail
      #"AV-30.22"(AUT_OP := wire#w1, LOCK := #"lock 2", ERR_EXTERN :=, LIOP_SEL := #init, L_AUT := #init, L_REMOTE := #init, L_SIM :=, L_RESET := #reset, MAN_OP :=, SIM_OP :=, FB_OPEN :=, FB_CLOSE :=, L_MON := #init, MON_T :=, MON_T_CLOSE :=, INSTANCE := 'AV-30.22', RESTART :=, VISIBILITY :=, OPdwCmd :=, QdwState =>, QwState =>, QCLOSING =>, QCLOSE =>, QOPENING =>, QOPEN =>, QCMD_OP => "AV-30.22", QMON =>, QMON_ERR =>, QMON_T =>, QMON_T_CLOSE =>, QMAN_AUT =>, QREMOTE =>, QSIM =>, QLOCK =>, QERR =>, QERR_EXT =>, QwAlarm =>)
   END_RUNG
   RUNG wire#powerrail
      Contact( "Blend_T-30".Out_AV_Header1 )
      Contact( "Blend_T-30"."HW Flushing".Status.Drain )
   END_RUNG wire#w1
   // the same network as SCL:
   #"AV-30.22"(LOCK := #"lock 2",   // "Valve"
               LIOP_SEL := #init,
               L_AUT := #init,
               L_REMOTE := #init,
               L_RESET := #reset,
               AUT_OP := "Blend_T-30".Out_AV_Header1 AND "Blend_T-30"."HW Flushing".Status.Drain,
               L_MON := #init,
               INSTANCE := 'AV-30.22',
               QCMD_OP => "AV-30.22");
END_REGION

REGION Network 26: AV-30.23 w ZSC
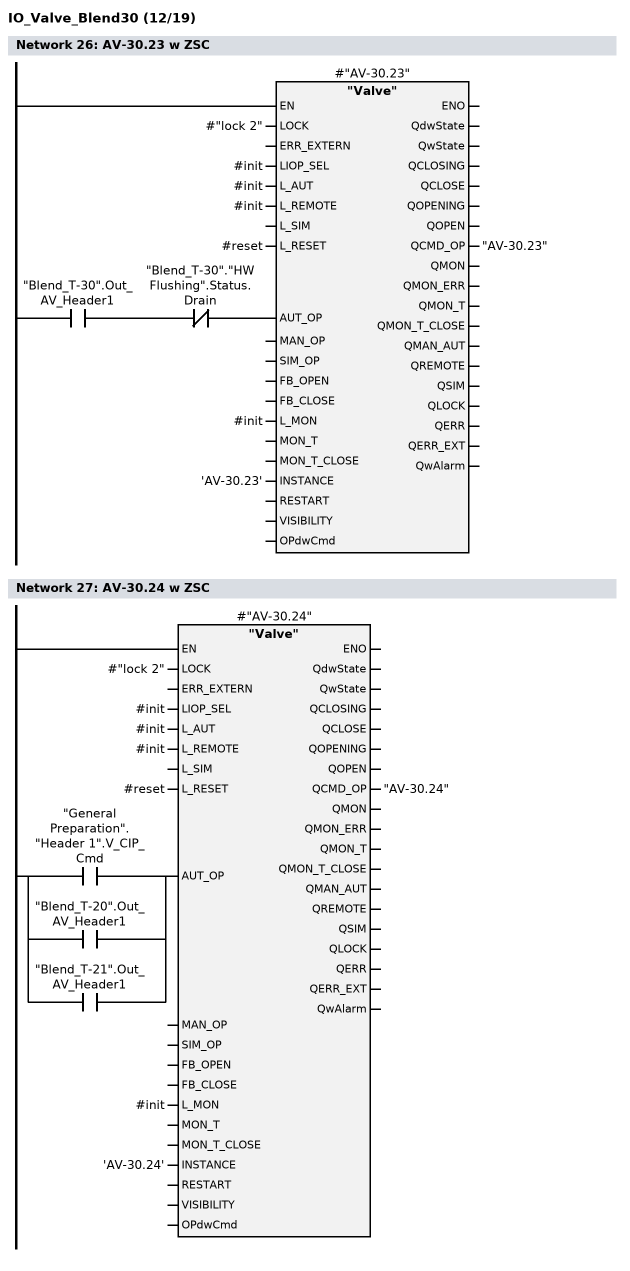
   RUNG wire#powerrail
      #"AV-30.23"(AUT_OP := wire#w1, LOCK := #"lock 2", ERR_EXTERN :=, LIOP_SEL := #init, L_AUT := #init, L_REMOTE := #init, L_SIM :=, L_RESET := #reset, MAN_OP :=, SIM_OP :=, FB_OPEN :=, FB_CLOSE :=, L_MON := #init, MON_T :=, MON_T_CLOSE :=, INSTANCE := 'AV-30.23', RESTART :=, VISIBILITY :=, OPdwCmd :=, QdwState =>, QwState =>, QCLOSING =>, QCLOSE =>, QOPENING =>, QOPEN =>, QCMD_OP => "AV-30.23", QMON =>, QMON_ERR =>, QMON_T =>, QMON_T_CLOSE =>, QMAN_AUT =>, QREMOTE =>, QSIM =>, QLOCK =>, QERR =>, QERR_EXT =>, QwAlarm =>)
   END_RUNG
   RUNG wire#powerrail
      Contact( "Blend_T-30".Out_AV_Header1 )
      I_Contact( "Blend_T-30"."HW Flushing".Status.Drain )
   END_RUNG wire#w1
   // the same network as SCL:
   #"AV-30.23"(LOCK := #"lock 2",   // "Valve"
               LIOP_SEL := #init,
               L_AUT := #init,
               L_REMOTE := #init,
               L_RESET := #reset,
               AUT_OP := "Blend_T-30".Out_AV_Header1 AND NOT "Blend_T-30"."HW Flushing".Status.Drain,
               L_MON := #init,
               INSTANCE := 'AV-30.23',
               QCMD_OP => "AV-30.23");
END_REGION

REGION Network 27: AV-30.24 w ZSC
   RUNG wire#powerrail
      #"AV-30.24"(AUT_OP := wire#w1, LOCK := #"lock 2", ERR_EXTERN :=, LIOP_SEL := #init, L_AUT := #init, L_REMOTE := #init, L_SIM :=, L_RESET := #reset, MAN_OP :=, SIM_OP :=, FB_OPEN :=, FB_CLOSE :=, L_MON := #init, MON_T :=, MON_T_CLOSE :=, INSTANCE := 'AV-30.24', RESTART :=, VISIBILITY :=, OPdwCmd :=, QdwState =>, QwState =>, QCLOSING =>, QCLOSE =>, QOPENING =>, QOPEN =>, QCMD_OP => "AV-30.24", QMON =>, QMON_ERR =>, QMON_T =>, QMON_T_CLOSE =>, QMAN_AUT =>, QREMOTE =>, QSIM =>, QLOCK =>, QERR =>, QERR_EXT =>, QwAlarm =>)
   END_RUNG
   RUNG wire#powerrail
      Contact( "General Preparation"."Header 1".V_CIP_Cmd )
   END_RUNG wire#w1
   RUNG wire#powerrail
      Contact( "Blend_T-20".Out_AV_Header1 )
   END_RUNG wire#w1
   RUNG wire#powerrail
      Contact( "Blend_T-21".Out_AV_Header1 )
   END_RUNG wire#w1
   // the same network as SCL:
   #"AV-30.24"(LOCK := #"lock 2",   // "Valve"
               LIOP_SEL := #init,
               L_AUT := #init,
               L_REMOTE := #init,
               L_RESET := #reset,
               AUT_OP := "General Preparation"."Header 1".V_CIP_Cmd OR "Blend_T-20".Out_AV_Header1 OR "Blend_T-21".Out_AV_Header1,
               L_MON := #init,
               INSTANCE := 'AV-30.24',
               QCMD_OP => "AV-30.24");
END_REGION

REGION Network 28: AV-30.25 w ZSC
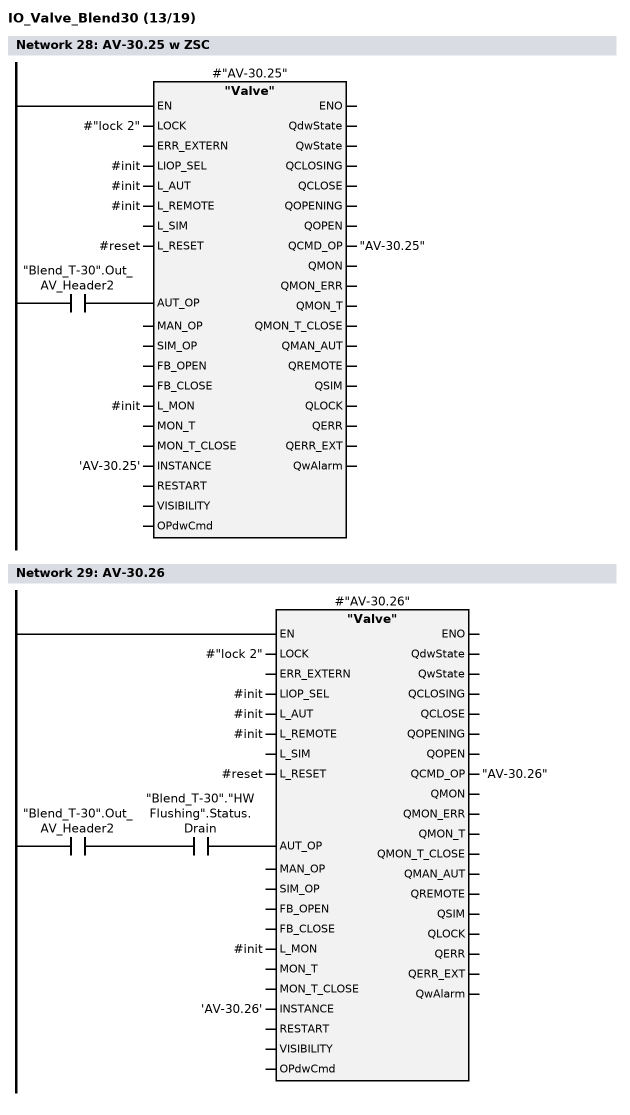
   RUNG wire#powerrail
      #"AV-30.25"(AUT_OP := wire#w1, LOCK := #"lock 2", ERR_EXTERN :=, LIOP_SEL := #init, L_AUT := #init, L_REMOTE := #init, L_SIM :=, L_RESET := #reset, MAN_OP :=, SIM_OP :=, FB_OPEN :=, FB_CLOSE :=, L_MON := #init, MON_T :=, MON_T_CLOSE :=, INSTANCE := 'AV-30.25', RESTART :=, VISIBILITY :=, OPdwCmd :=, QdwState =>, QwState =>, QCLOSING =>, QCLOSE =>, QOPENING =>, QOPEN =>, QCMD_OP => "AV-30.25", QMON =>, QMON_ERR =>, QMON_T =>, QMON_T_CLOSE =>, QMAN_AUT =>, QREMOTE =>, QSIM =>, QLOCK =>, QERR =>, QERR_EXT =>, QwAlarm =>)
   END_RUNG
   RUNG wire#powerrail
      Contact( "Blend_T-30".Out_AV_Header2 )
   END_RUNG wire#w1
   // the same network as SCL:
   #"AV-30.25"(LOCK := #"lock 2",   // "Valve"
               LIOP_SEL := #init,
               L_AUT := #init,
               L_REMOTE := #init,
               L_RESET := #reset,
               AUT_OP := "Blend_T-30".Out_AV_Header2,
               L_MON := #init,
               INSTANCE := 'AV-30.25',
               QCMD_OP => "AV-30.25");
END_REGION

REGION Network 29: AV-30.26
   RUNG wire#powerrail
      #"AV-30.26"(AUT_OP := wire#w1, LOCK := #"lock 2", ERR_EXTERN :=, LIOP_SEL := #init, L_AUT := #init, L_REMOTE := #init, L_SIM :=, L_RESET := #reset, MAN_OP :=, SIM_OP :=, FB_OPEN :=, FB_CLOSE :=, L_MON := #init, MON_T :=, MON_T_CLOSE :=, INSTANCE := 'AV-30.26', RESTART :=, VISIBILITY :=, OPdwCmd :=, QdwState =>, QwState =>, QCLOSING =>, QCLOSE =>, QOPENING =>, QOPEN =>, QCMD_OP => "AV-30.26", QMON =>, QMON_ERR =>, QMON_T =>, QMON_T_CLOSE =>, QMAN_AUT =>, QREMOTE =>, QSIM =>, QLOCK =>, QERR =>, QERR_EXT =>, QwAlarm =>)
   END_RUNG
   RUNG wire#powerrail
      Contact( "Blend_T-30".Out_AV_Header2 )
      Contact( "Blend_T-30"."HW Flushing".Status.Drain )
   END_RUNG wire#w1
   // the same network as SCL:
   #"AV-30.26"(LOCK := #"lock 2",   // "Valve"
               LIOP_SEL := #init,
               L_AUT := #init,
               L_REMOTE := #init,
               L_RESET := #reset,
               AUT_OP := "Blend_T-30".Out_AV_Header2 AND "Blend_T-30"."HW Flushing".Status.Drain,
               L_MON := #init,
               INSTANCE := 'AV-30.26',
               QCMD_OP => "AV-30.26");
END_REGION

REGION Network 30: AV-30.27 w ZSC
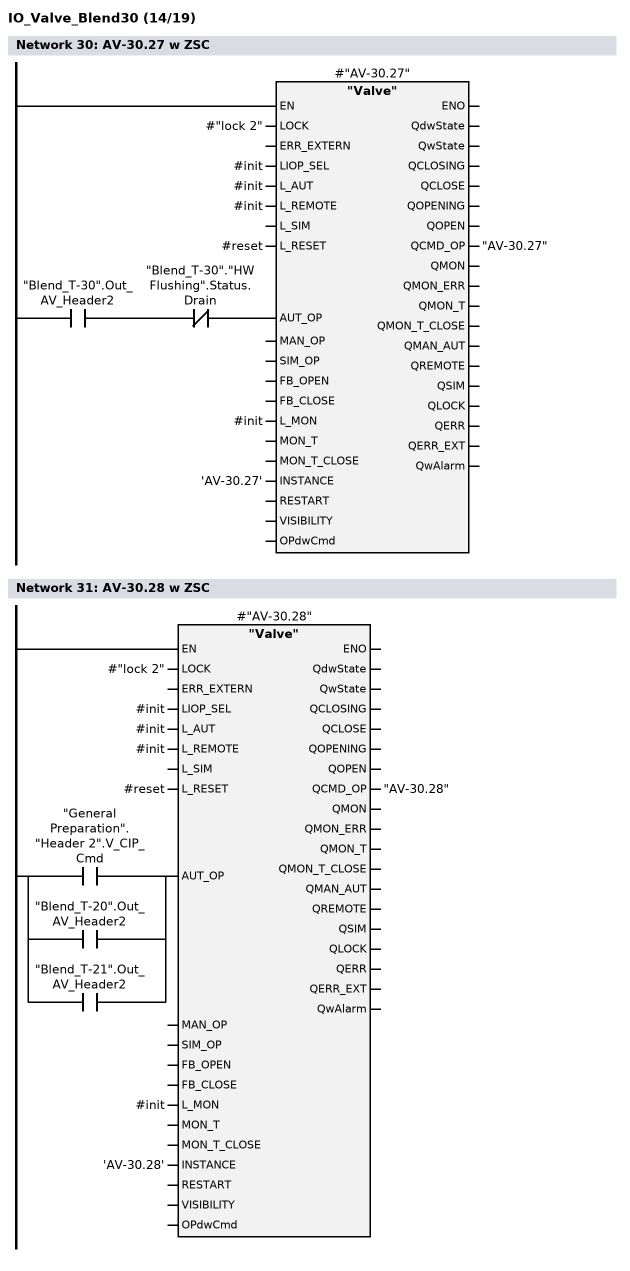
   RUNG wire#powerrail
      #"AV-30.27"(AUT_OP := wire#w1, LOCK := #"lock 2", ERR_EXTERN :=, LIOP_SEL := #init, L_AUT := #init, L_REMOTE := #init, L_SIM :=, L_RESET := #reset, MAN_OP :=, SIM_OP :=, FB_OPEN :=, FB_CLOSE :=, L_MON := #init, MON_T :=, MON_T_CLOSE :=, INSTANCE := 'AV-30.27', RESTART :=, VISIBILITY :=, OPdwCmd :=, QdwState =>, QwState =>, QCLOSING =>, QCLOSE =>, QOPENING =>, QOPEN =>, QCMD_OP => "AV-30.27", QMON =>, QMON_ERR =>, QMON_T =>, QMON_T_CLOSE =>, QMAN_AUT =>, QREMOTE =>, QSIM =>, QLOCK =>, QERR =>, QERR_EXT =>, QwAlarm =>)
   END_RUNG
   RUNG wire#powerrail
      Contact( "Blend_T-30".Out_AV_Header2 )
      I_Contact( "Blend_T-30"."HW Flushing".Status.Drain )
   END_RUNG wire#w1
   // the same network as SCL:
   #"AV-30.27"(LOCK := #"lock 2",   // "Valve"
               LIOP_SEL := #init,
               L_AUT := #init,
               L_REMOTE := #init,
               L_RESET := #reset,
               AUT_OP := "Blend_T-30".Out_AV_Header2 AND NOT "Blend_T-30"."HW Flushing".Status.Drain,
               L_MON := #init,
               INSTANCE := 'AV-30.27',
               QCMD_OP => "AV-30.27");
END_REGION

REGION Network 31: AV-30.28 w ZSC
   RUNG wire#powerrail
      #"AV-30.28"(AUT_OP := wire#w1, LOCK := #"lock 2", ERR_EXTERN :=, LIOP_SEL := #init, L_AUT := #init, L_REMOTE := #init, L_SIM :=, L_RESET := #reset, MAN_OP :=, SIM_OP :=, FB_OPEN :=, FB_CLOSE :=, L_MON := #init, MON_T :=, MON_T_CLOSE :=, INSTANCE := 'AV-30.28', RESTART :=, VISIBILITY :=, OPdwCmd :=, QdwState =>, QwState =>, QCLOSING =>, QCLOSE =>, QOPENING =>, QOPEN =>, QCMD_OP => "AV-30.28", QMON =>, QMON_ERR =>, QMON_T =>, QMON_T_CLOSE =>, QMAN_AUT =>, QREMOTE =>, QSIM =>, QLOCK =>, QERR =>, QERR_EXT =>, QwAlarm =>)
   END_RUNG
   RUNG wire#powerrail
      Contact( "General Preparation"."Header 2".V_CIP_Cmd )
   END_RUNG wire#w1
   RUNG wire#powerrail
      Contact( "Blend_T-20".Out_AV_Header2 )
   END_RUNG wire#w1
   RUNG wire#powerrail
      Contact( "Blend_T-21".Out_AV_Header2 )
   END_RUNG wire#w1
   // the same network as SCL:
   #"AV-30.28"(LOCK := #"lock 2",   // "Valve"
               LIOP_SEL := #init,
               L_AUT := #init,
               L_REMOTE := #init,
               L_RESET := #reset,
               AUT_OP := "General Preparation"."Header 2".V_CIP_Cmd OR "Blend_T-20".Out_AV_Header2 OR "Blend_T-21".Out_AV_Header2,
               L_MON := #init,
               INSTANCE := 'AV-30.28',
               QCMD_OP => "AV-30.28");
END_REGION

REGION Network 32: AV-30.29
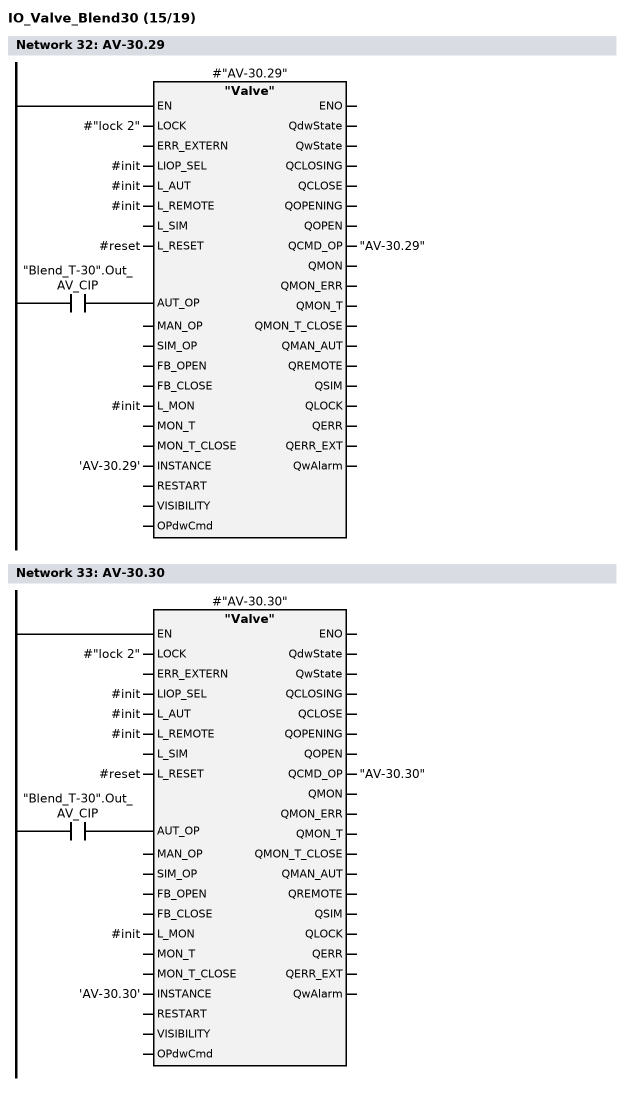
   RUNG wire#powerrail
      #"AV-30.29"(AUT_OP := wire#w1, LOCK := #"lock 2", ERR_EXTERN :=, LIOP_SEL := #init, L_AUT := #init, L_REMOTE := #init, L_SIM :=, L_RESET := #reset, MAN_OP :=, SIM_OP :=, FB_OPEN :=, FB_CLOSE :=, L_MON := #init, MON_T :=, MON_T_CLOSE :=, INSTANCE := 'AV-30.29', RESTART :=, VISIBILITY :=, OPdwCmd :=, QdwState =>, QwState =>, QCLOSING =>, QCLOSE =>, QOPENING =>, QOPEN =>, QCMD_OP => "AV-30.29", QMON =>, QMON_ERR =>, QMON_T =>, QMON_T_CLOSE =>, QMAN_AUT =>, QREMOTE =>, QSIM =>, QLOCK =>, QERR =>, QERR_EXT =>, QwAlarm =>)
   END_RUNG
   RUNG wire#powerrail
      Contact( "Blend_T-30".Out_AV_CIP )
   END_RUNG wire#w1
   // the same network as SCL:
   #"AV-30.29"(LOCK := #"lock 2",   // "Valve"
               LIOP_SEL := #init,
               L_AUT := #init,
               L_REMOTE := #init,
               L_RESET := #reset,
               AUT_OP := "Blend_T-30".Out_AV_CIP,
               L_MON := #init,
               INSTANCE := 'AV-30.29',
               QCMD_OP => "AV-30.29");
END_REGION

REGION Network 33: AV-30.30
   RUNG wire#powerrail
      #"AV-30.30"(AUT_OP := wire#w1, LOCK := #"lock 2", ERR_EXTERN :=, LIOP_SEL := #init, L_AUT := #init, L_REMOTE := #init, L_SIM :=, L_RESET := #reset, MAN_OP :=, SIM_OP :=, FB_OPEN :=, FB_CLOSE :=, L_MON := #init, MON_T :=, MON_T_CLOSE :=, INSTANCE := 'AV-30.30', RESTART :=, VISIBILITY :=, OPdwCmd :=, QdwState =>, QwState =>, QCLOSING =>, QCLOSE =>, QOPENING =>, QOPEN =>, QCMD_OP => "AV-30.30", QMON =>, QMON_ERR =>, QMON_T =>, QMON_T_CLOSE =>, QMAN_AUT =>, QREMOTE =>, QSIM =>, QLOCK =>, QERR =>, QERR_EXT =>, QwAlarm =>)
   END_RUNG
   RUNG wire#powerrail
      Contact( "Blend_T-30".Out_AV_CIP )
   END_RUNG wire#w1
   // the same network as SCL:
   #"AV-30.30"(LOCK := #"lock 2",   // "Valve"
               LIOP_SEL := #init,
               L_AUT := #init,
               L_REMOTE := #init,
               L_RESET := #reset,
               AUT_OP := "Blend_T-30".Out_AV_CIP,
               L_MON := #init,
               INSTANCE := 'AV-30.30',
               QCMD_OP => "AV-30.30");
END_REGION

REGION Network 34: AV-30.31 w ZSC
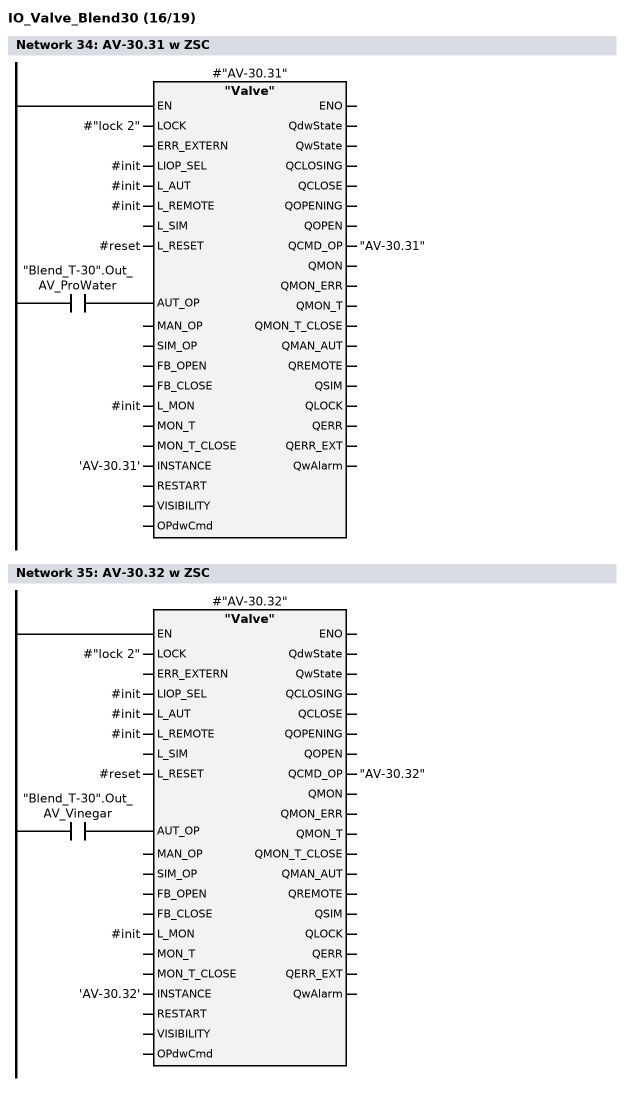
   RUNG wire#powerrail
      #"AV-30.31"(AUT_OP := wire#w1, LOCK := #"lock 2", ERR_EXTERN :=, LIOP_SEL := #init, L_AUT := #init, L_REMOTE := #init, L_SIM :=, L_RESET := #reset, MAN_OP :=, SIM_OP :=, FB_OPEN :=, FB_CLOSE :=, L_MON := #init, MON_T :=, MON_T_CLOSE :=, INSTANCE := 'AV-30.31', RESTART :=, VISIBILITY :=, OPdwCmd :=, QdwState =>, QwState =>, QCLOSING =>, QCLOSE =>, QOPENING =>, QOPEN =>, QCMD_OP => "AV-30.31", QMON =>, QMON_ERR =>, QMON_T =>, QMON_T_CLOSE =>, QMAN_AUT =>, QREMOTE =>, QSIM =>, QLOCK =>, QERR =>, QERR_EXT =>, QwAlarm =>)
   END_RUNG
   RUNG wire#powerrail
      Contact( "Blend_T-30".Out_AV_ProWater )
   END_RUNG wire#w1
   // the same network as SCL:
   #"AV-30.31"(LOCK := #"lock 2",   // "Valve"
               LIOP_SEL := #init,
               L_AUT := #init,
               L_REMOTE := #init,
               L_RESET := #reset,
               AUT_OP := "Blend_T-30".Out_AV_ProWater,
               L_MON := #init,
               INSTANCE := 'AV-30.31',
               QCMD_OP => "AV-30.31");
END_REGION

REGION Network 35: AV-30.32 w ZSC
   RUNG wire#powerrail
      #"AV-30.32"(AUT_OP := wire#w1, LOCK := #"lock 2", ERR_EXTERN :=, LIOP_SEL := #init, L_AUT := #init, L_REMOTE := #init, L_SIM :=, L_RESET := #reset, MAN_OP :=, SIM_OP :=, FB_OPEN :=, FB_CLOSE :=, L_MON := #init, MON_T :=, MON_T_CLOSE :=, INSTANCE := 'AV-30.32', RESTART :=, VISIBILITY :=, OPdwCmd :=, QdwState =>, QwState =>, QCLOSING =>, QCLOSE =>, QOPENING =>, QOPEN =>, QCMD_OP => "AV-30.32", QMON =>, QMON_ERR =>, QMON_T =>, QMON_T_CLOSE =>, QMAN_AUT =>, QREMOTE =>, QSIM =>, QLOCK =>, QERR =>, QERR_EXT =>, QwAlarm =>)
   END_RUNG
   RUNG wire#powerrail
      Contact( "Blend_T-30".Out_AV_Vinegar )
   END_RUNG wire#w1
   // the same network as SCL:
   #"AV-30.32"(LOCK := #"lock 2",   // "Valve"
               LIOP_SEL := #init,
               L_AUT := #init,
               L_REMOTE := #init,
               L_RESET := #reset,
               AUT_OP := "Blend_T-30".Out_AV_Vinegar,
               L_MON := #init,
               INSTANCE := 'AV-30.32',
               QCMD_OP => "AV-30.32");
END_REGION

REGION Network 36: AV-30.33 w ZSC
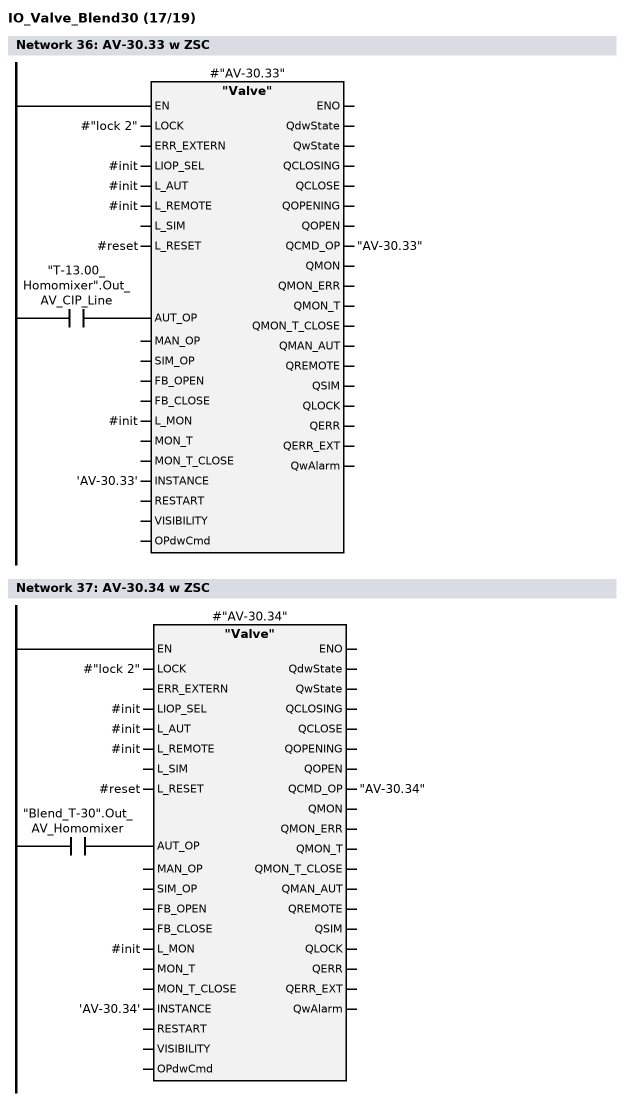
   RUNG wire#powerrail
      #"AV-30.33"(AUT_OP := wire#w1, LOCK := #"lock 2", ERR_EXTERN :=, LIOP_SEL := #init, L_AUT := #init, L_REMOTE := #init, L_SIM :=, L_RESET := #reset, MAN_OP :=, SIM_OP :=, FB_OPEN :=, FB_CLOSE :=, L_MON := #init, MON_T :=, MON_T_CLOSE :=, INSTANCE := 'AV-30.33', RESTART :=, VISIBILITY :=, OPdwCmd :=, QdwState =>, QwState =>, QCLOSING =>, QCLOSE =>, QOPENING =>, QOPEN =>, QCMD_OP => "AV-30.33", QMON =>, QMON_ERR =>, QMON_T =>, QMON_T_CLOSE =>, QMAN_AUT =>, QREMOTE =>, QSIM =>, QLOCK =>, QERR =>, QERR_EXT =>, QwAlarm =>)
   END_RUNG
   RUNG wire#powerrail
      Contact( "T-13.00_Homomixer".Out_AV_CIP_Line )
   END_RUNG wire#w1
   // the same network as SCL:
   #"AV-30.33"(LOCK := #"lock 2",   // "Valve"
               LIOP_SEL := #init,
               L_AUT := #init,
               L_REMOTE := #init,
               L_RESET := #reset,
               AUT_OP := "T-13.00_Homomixer".Out_AV_CIP_Line,
               L_MON := #init,
               INSTANCE := 'AV-30.33',
               QCMD_OP => "AV-30.33");
END_REGION

REGION Network 37: AV-30.34 w ZSC
   RUNG wire#powerrail
      #"AV-30.34"(AUT_OP := wire#w1, LOCK := #"lock 2", ERR_EXTERN :=, LIOP_SEL := #init, L_AUT := #init, L_REMOTE := #init, L_SIM :=, L_RESET := #reset, MAN_OP :=, SIM_OP :=, FB_OPEN :=, FB_CLOSE :=, L_MON := #init, MON_T :=, MON_T_CLOSE :=, INSTANCE := 'AV-30.34', RESTART :=, VISIBILITY :=, OPdwCmd :=, QdwState =>, QwState =>, QCLOSING =>, QCLOSE =>, QOPENING =>, QOPEN =>, QCMD_OP => "AV-30.34", QMON =>, QMON_ERR =>, QMON_T =>, QMON_T_CLOSE =>, QMAN_AUT =>, QREMOTE =>, QSIM =>, QLOCK =>, QERR =>, QERR_EXT =>, QwAlarm =>)
   END_RUNG
   RUNG wire#powerrail
      Contact( "Blend_T-30".Out_AV_Homomixer )
   END_RUNG wire#w1
   // the same network as SCL:
   #"AV-30.34"(LOCK := #"lock 2",   // "Valve"
               LIOP_SEL := #init,
               L_AUT := #init,
               L_REMOTE := #init,
               L_RESET := #reset,
               AUT_OP := "Blend_T-30".Out_AV_Homomixer,
               L_MON := #init,
               INSTANCE := 'AV-30.34',
               QCMD_OP => "AV-30.34");
END_REGION

REGION Network 38: AV-30.35 w ZSC
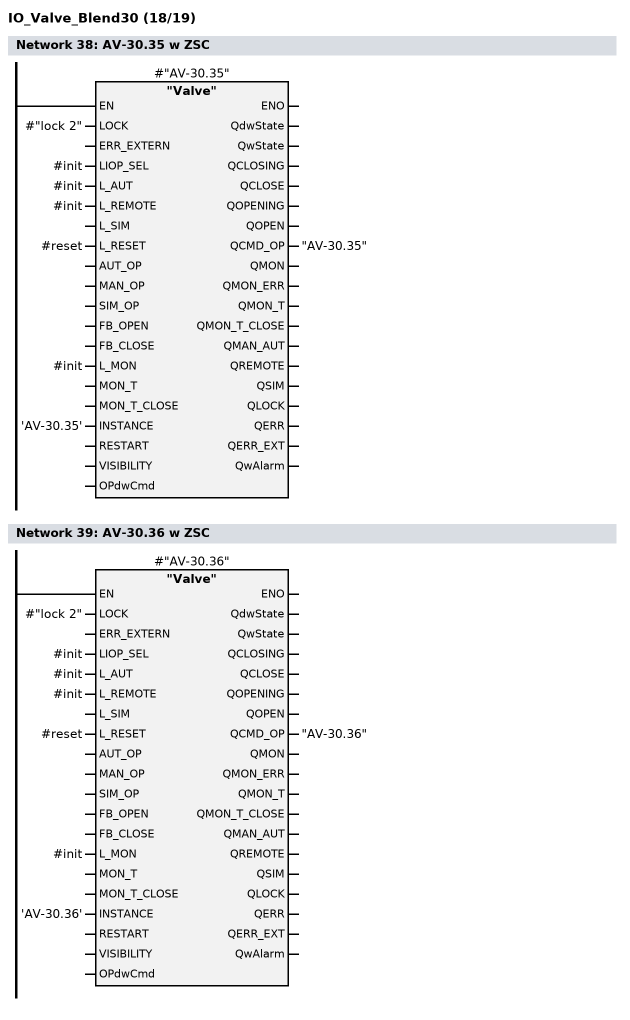
   RUNG wire#powerrail
      #"AV-30.35"(LOCK := #"lock 2", ERR_EXTERN :=, LIOP_SEL := #init, L_AUT := #init, L_REMOTE := #init, L_SIM :=, L_RESET := #reset, AUT_OP :=, MAN_OP :=, SIM_OP :=, FB_OPEN :=, FB_CLOSE :=, L_MON := #init, MON_T :=, MON_T_CLOSE :=, INSTANCE := 'AV-30.35', RESTART :=, VISIBILITY :=, OPdwCmd :=, QdwState =>, QwState =>, QCLOSING =>, QCLOSE =>, QOPENING =>, QOPEN =>, QCMD_OP => "AV-30.35", QMON =>, QMON_ERR =>, QMON_T =>, QMON_T_CLOSE =>, QMAN_AUT =>, QREMOTE =>, QSIM =>, QLOCK =>, QERR =>, QERR_EXT =>, QwAlarm =>)
   END_RUNG
   // the same network as SCL:
   #"AV-30.35"(LOCK := #"lock 2",   // "Valve"
               LIOP_SEL := #init,
               L_AUT := #init,
               L_REMOTE := #init,
               L_RESET := #reset,
               L_MON := #init,
               INSTANCE := 'AV-30.35',
               QCMD_OP => "AV-30.35");
END_REGION

REGION Network 39: AV-30.36 w ZSC
   RUNG wire#powerrail
      #"AV-30.36"(LOCK := #"lock 2", ERR_EXTERN :=, LIOP_SEL := #init, L_AUT := #init, L_REMOTE := #init, L_SIM :=, L_RESET := #reset, AUT_OP :=, MAN_OP :=, SIM_OP :=, FB_OPEN :=, FB_CLOSE :=, L_MON := #init, MON_T :=, MON_T_CLOSE :=, INSTANCE := 'AV-30.36', RESTART :=, VISIBILITY :=, OPdwCmd :=, QdwState =>, QwState =>, QCLOSING =>, QCLOSE =>, QOPENING =>, QOPEN =>, QCMD_OP => "AV-30.36", QMON =>, QMON_ERR =>, QMON_T =>, QMON_T_CLOSE =>, QMAN_AUT =>, QREMOTE =>, QSIM =>, QLOCK =>, QERR =>, QERR_EXT =>, QwAlarm =>)
   END_RUNG
   // the same network as SCL:
   #"AV-30.36"(LOCK := #"lock 2",   // "Valve"
               LIOP_SEL := #init,
               L_AUT := #init,
               L_REMOTE := #init,
               L_RESET := #reset,
               L_MON := #init,
               INSTANCE := 'AV-30.36',
               QCMD_OP => "AV-30.36");
END_REGION

REGION Network 40: AV-30.41
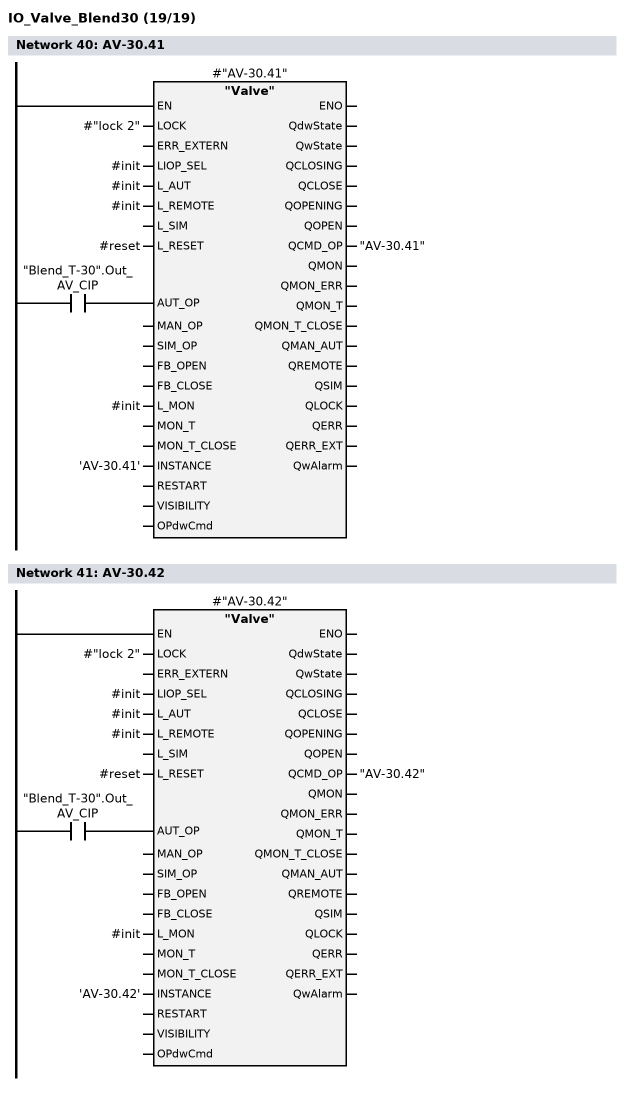
   RUNG wire#powerrail
      #"AV-30.41"(AUT_OP := wire#w1, LOCK := #"lock 2", ERR_EXTERN :=, LIOP_SEL := #init, L_AUT := #init, L_REMOTE := #init, L_SIM :=, L_RESET := #reset, MAN_OP :=, SIM_OP :=, FB_OPEN :=, FB_CLOSE :=, L_MON := #init, MON_T :=, MON_T_CLOSE :=, INSTANCE := 'AV-30.41', RESTART :=, VISIBILITY :=, OPdwCmd :=, QdwState =>, QwState =>, QCLOSING =>, QCLOSE =>, QOPENING =>, QOPEN =>, QCMD_OP => "AV-30.41", QMON =>, QMON_ERR =>, QMON_T =>, QMON_T_CLOSE =>, QMAN_AUT =>, QREMOTE =>, QSIM =>, QLOCK =>, QERR =>, QERR_EXT =>, QwAlarm =>)
   END_RUNG
   RUNG wire#powerrail
      Contact( "Blend_T-30".Out_AV_CIP )
   END_RUNG wire#w1
   // the same network as SCL:
   #"AV-30.41"(LOCK := #"lock 2",   // "Valve"
               LIOP_SEL := #init,
               L_AUT := #init,
               L_REMOTE := #init,
               L_RESET := #reset,
               AUT_OP := "Blend_T-30".Out_AV_CIP,
               L_MON := #init,
               INSTANCE := 'AV-30.41',
               QCMD_OP => "AV-30.41");
END_REGION

REGION Network 41: AV-30.42
   RUNG wire#powerrail
      #"AV-30.42"(AUT_OP := wire#w1, LOCK := #"lock 2", ERR_EXTERN :=, LIOP_SEL := #init, L_AUT := #init, L_REMOTE := #init, L_SIM :=, L_RESET := #reset, MAN_OP :=, SIM_OP :=, FB_OPEN :=, FB_CLOSE :=, L_MON := #init, MON_T :=, MON_T_CLOSE :=, INSTANCE := 'AV-30.42', RESTART :=, VISIBILITY :=, OPdwCmd :=, QdwState =>, QwState =>, QCLOSING =>, QCLOSE =>, QOPENING =>, QOPEN =>, QCMD_OP => "AV-30.42", QMON =>, QMON_ERR =>, QMON_T =>, QMON_T_CLOSE =>, QMAN_AUT =>, QREMOTE =>, QSIM =>, QLOCK =>, QERR =>, QERR_EXT =>, QwAlarm =>)
   END_RUNG
   RUNG wire#powerrail
      Contact( "Blend_T-30".Out_AV_CIP )
   END_RUNG wire#w1
   // the same network as SCL:
   #"AV-30.42"(LOCK := #"lock 2",   // "Valve"
               LIOP_SEL := #init,
               L_AUT := #init,
               L_REMOTE := #init,
               L_RESET := #reset,
               AUT_OP := "Blend_T-30".Out_AV_CIP,
               L_MON := #init,
               INSTANCE := 'AV-30.42',
               QCMD_OP => "AV-30.42");
END_REGION
END_FUNCTION_BLOCK
